// SIMATIC STEP 7 (V5.x) project PlcTornioFisher
// CPU: PLC317-2DP
// station: Hardware
// station: SINUMERIK
// station: P_ADR_BUS
// program: Programma S7(1)
// program: gp8x0d - PLC-Basicprogram-800Dsl 02.07.06 11/08/15
// program: SINAMICS_In_NCU_720
// program: SINAMICS_NX15_SINUMERIK

SYMBOL_TABLE
"ALMSG_DB"	DB 2	UDT 2	// Interface for Alarms & Messages
"gp_par"	DB 7	FB 1	// Parameters for Baseprogram
"NC"	DB 10	UDT 10	// Interface NC
"BAG"	DB 11	UDT 11	// Interface for BAG
"PI"	DB 16	DB 16	// Datainterface PI-Services
"SPL"	DB 18	DB 18	// SPL dataarea
"MMC"	DB 19	UDT 19	// Interface MMC-Signals
"Opzioni"	DB 20	UDT 20	// Opzioni macchina
"Canale1"	DB 21	UDT 21	// Interfaccia per Canale 1
"Canale2"	DB 22	UDT 21	// Interfaccia per Canale 2
"Canale3"	DB 23	UDT 21	// Interfaccia per Canale 3
"Canale4"	DB 24	UDT 21	// Interfaccia per Canale 4
"Asse_X1"	DB 31	UDT 31	// Interfaccia per Asse X1
"Asse_Z1"	DB 32	UDT 31	// Interfaccia per Asse Z1
"Asse_A"	DB 33	UDT 31	// Interfaccia per Asse A
"Asse_X2"	DB 34	UDT 31	// Interfaccia per Asse X2
"Asse_Z2"	DB 35	UDT 31	// Interfaccia per Asse Z2
"Asse_B"	DB 36	UDT 31	// Interfaccia per Asse B
"Asse_W"	DB 37	UDT 31	// Interfaccia per Asse W
"Asse_SP"	DB 38	UDT 31	// Interfaccia per Mandrino
"TMLoadIF"	DB 71	UDT 71	// Interface for Loading Station (Toolmanag.)
"TMSpindleIF"	DB 72	UDT 72	// Interface Spindle for Toolmanagment
"TMRevIF"	DB 73	UDT 73	// Interface Revolver (Toolmanagment)
"DB77"	DB 77	UDT 77	// SIEMENS
"CtrlE"	DB 1000	DB 1000	// Interface Ctrl-Energy
"SentronPac"	DB 1001	DB 1001	// Interface SentronPac
"RUN_UP"	FB 1	FB 1	// Startup Baseprogram
"GET"	FB 2	FB 2	// read NC Variable
"PUT"	FB 3	FB 3	// write NC Variable
"PI_SERV"	FB 4	FB 4	// PI-Services 1
"GETGUD"	FB 5	FB 5	// read GUD-Variable
"PI_SERV2"	FB 7	FB 7	// PI-Services 2
"M2N"	FB 9	FB 9	// Several OPs/NCUs
"SI_Relais"	FB 10	FB 10	// Safety Integrated: Relais
"SI_BrakeTest"	FB 11	FB 11	// Safety Integrated: Brake Test
"Diagnose"	FB 29	FB 29	// Signal recorder and data trigger diagnostics
"GP_HP"	FC 2	FC 2	// cyclic Baseprogram
"GP_PRAL"	FC 3	FC 3	// alarmtriggered Baseprogram
"GP_DIAG"	FC 5	FC 5	// Diagnosis alarm and Modul failure
"TM_TRANS2"	FC 6	FC 6	// Transfer for Toolmanagment (Multitool)
"TM_REV"	FC 7	FC 7	// Transfer for Revolverchange
"TM_TRANS"	FC 8	FC 8	// Transfer for Toolmanagment
"ASUP"	FC 9	FC 9	// asynchronous Subprograms
"AL_MSG"	FC 10	FC 10	// Alarms & Messages
"BHGDisp"	FC 13	FC 13	// Displaycontrol for Handheld Unit
"YDelta"	FC 17	FC 17	// Y / Delta Control
"SpinCtrl"	FC 18	FC 18	// Spindlecontrol / Part-, Positioning-axis
"MCP_IFM"	FC 19	FC 19	// MCP-Signals to Interface, Variant M
"Transfer"	FC 21	FC 21	// Quick Datachannel
"TM_DIR"	FC 22	FC 22	// Directioncontrol for Toolmanagment Mag.
"MCP_IFM2"	FC 24	FC 24	// MCP-Signals to Interface, Variant small
"MCP_IFT"	FC 25	FC 25	// MCP-Signals to Interface, Variant T
"HPU_MCP"	FC 26	FC 26	// MCP-Signals of PHG to Interface
"iNO_Emergenza_C1"	I 32.0	BOOL	// Emergenza ripristinata (Canale 1)
"iAux_ON(NC)"	I 32.1	BOOL	// Ausiliari inseriti (NC)
"iMax_Temp_AR"	I 32.2	BOOL	// Max temperatura alimentatore assi e mandrino
"iAR_Pronto"	I 32.3	BOOL	// Alimentatore assi e mandrino pronto
"iMax_Temp_Sorvegl"	I 32.4	BOOL	// Max temperatura modulo di sorveglianza
"iSorvegl_Pronto"	I 32.5	BOOL	// Modulo di sorveglianza pronto
"iPuls_Consenso"	I 32.6	BOOL	// 20SB1 - 20KA1 - Pulsante di consenso
"iAux_ON(NA)"	I 32.7	BOOL	// 18KA1 - Ausiliari inseriti (NA)
"iQM_Pompa_Idraul"	I 33.0	BOOL	// 3QM1 - Magnetotermico Pompa idraulica
"iQM_Sist_Serraggio"	I 33.1	BOOL	// 3QM2 - Magnetotermico Sistema di serraggio
"iQM_Controllo_Utensili"	I 33.2	BOOL	// 3QM3 - Magnetotermico Dispositivo Controllo Utensili
"iQM_Ventilat_Mandrino"	I 33.3	BOOL	// 3QM4 - MagnetotermicoVentilatore Mandrino
"iQF_Trasformatore"	I 33.4	BOOL	// 4QF1 - Magnetotermico Protezione trasformatore
"iQF_Utenze_110Vac"	I 33.5	BOOL	// 4QF2 - Magnetotermico Protezione Utenze a 110 Vac
"iQF_Prese_Illuminaz_QE"	I 33.6	BOOL	// 4QF3+4QF4 - Magnetot. Protez. Presa Pulpito e Q.E. +Illuminaz. Quadro
"iQF_Montronix"	I 33.7	BOOL	// 4QF5 - Magnetotermico Protezione Alimentazione Montronix
"iQF_Alim_24V_Uscite"	I 34.0	BOOL	// 5QF1 - Magnetotermico Protezione Sitop 24V Uscite
"iQF_Illuminaz_Macch"	I 34.1	BOOL	// 5QF2 - Magnetotermico Protezione Illuminaz. Macchina
"iQF_24V_UsciteSempreAlim"	I 34.2	BOOL	// 5QF3 - Magnetotermico Protezione Uscite PLC sempre alimentate
"iQF_24V_Uscite_Sezionate"	I 34.3	BOOL	// 5QF4 - Magnetotermico Protezione Uscite PLC sezionate
"iQF_Marposs"	I 34.4	BOOL	// 5QF6 - Magnetotermico Protezione Marposs
"iQF_Elettronica_CN"	I 34.5	BOOL	// 5QF7 - Magnetotermico Protezione Elettronica CN
"iQF_Condizionatori"	I 34.6	BOOL	// 6QF1+6QF2 Magnetot. Protez. condizionatori e trasformatore condizionatori
"iQF_Freno_Mandrino"	I 34.7	BOOL	// 12QF1 - Magnetotermico Protezione Freno Mandrino
"iQF_Uscite_Caricatore"	I 35.0	BOOL	// 5QF8 - Magnetotermico Protezione Uscite Caricatore
"iQF_Ingressi_PLC"	I 35.1	BOOL	// 5QF5 - Magnetotermico Protezione Alimentazione Ingressi PLC
"iBP35.2"	I 35.2	BOOL	// BP35.2 - Pressostato Blocco utensili sistema B serrato
"iBP35.3"	I 35.3	BOOL	// BP35.3 - Pressostato Blocco utensili sistema B disserrato
"iBP35.4"	I 35.4	BOOL	// BP35.4 - Pressostato Blocco utensili sistema A serrato
"iBP35.5"	I 35.5	BOOL	// BP35.5 - Pressostato Blocco utensili sistema A disserrato
"iBQ_Rip_Renishaw_Chiuso"	I 35.6	BOOL	// BP35.6 - Proximity Riparo controllo utensili chiuso
"iBQ_Rip_Renishaw_Aperto"	I 35.7	BOOL	// BP35.7 - Proximity Riparo controllo utensili aperto
"iNO_Emergenza_C2"	I 36.0	BOOL	// Emergenza ripristinata (Canale 2)
"iSA_AUTO"	I 36.1	BOOL	// SA36.1 - Selettore Funzionamento automatico
"iBQ36.3"	I 36.3	BOOL	// BQ36.3 - Proximity Braccio di misura in posiz. di misura
"iBQ36.4"	I 36.4	BOOL	// BQ36.4 - Proximity Braccio di misura a riposo
"iBP36.5"	I 36.5	BOOL	// BQ36.5 - Pressostato Filtro serraggio OK
"iKM_Pompa_Oleod_Inserita"	I 36.6	BOOL	// 51KM1 - Pompa oleodinamica inserita
"E36.7"	I 36.7	BOOL	// Disponibile
"iSQ_Oltrecorsa_X1+"	I 37.0	BOOL	// SQ37.0 - Finecorsa Oltrecorsa asse X1+
"iSQ_Oltrecorsa_X1-"	I 37.1	BOOL	// SQ37.1 - Finecorsa Oltrecorsa asse X1-
"iSQ_Ref_X1"	I 37.2	BOOL	// SQ37.2 - Finecorsa Punto di riferimento asse X1
"iSQ_Oltrecorsa_Z1+"	I 37.3	BOOL	// SQ37.3 - Finecorsa Oltrecorsa asse Z1+
"iSQ_Oltrecorsa_Z1-"	I 37.4	BOOL	// SQ37.4 - Finecorsa Oltrecorsa asse Z1-
"iSQ_Ref_Z1"	I 37.5	BOOL	// SQ37.5 - Finecorsa Punto di riferimento asse Z1
"iSQ_Oltrecorsa_X2+"	I 37.6	BOOL	// SQ37.6 - Finecorsa Oltrecorsa asse X2+
"iSQ_Oltrecorsa_X2-"	I 37.7	BOOL	// SQ37.7 - Finecorsa Oltrecorsa asse X2-
"iSQ_Ref_X2"	I 38.0	BOOL	// SQ38.0 - Finecorsa Punto di riferimento asse X2
"iSQ_Oltrecorsa_Z2+"	I 38.1	BOOL	// SQ38.1 - Finecorsa Oltrecorsa asse Z2+
"iSQ_Oltrecorsa_Z2-"	I 38.2	BOOL	// SQ38.2 - Finecorsa Oltrecorsa  asse Z2-
"iSQ_Ref_Z2_A"	I 38.3	BOOL	// SQ38.3 - Finecorsa Punto di riferimento A asse Z2
"iSQ_Ref_Z2_B"	I 38.4	BOOL	// SQ38.4 - Finecorsa Punto di riferimento B asse Z2
"iSQ_Cann_Avanz"	I 38.5	BOOL	// SQ38.5 - Finecorsa Posizione Cannotto Avanzato
"iSQ_Cann_Richiam"	I 38.6	BOOL	// SQ38.6 - Finecorsa Posizione Cannotto Richiamato
"iSQ_Oltrecorsa_W+"	I 38.7	BOOL	// SQ38.7 - Finecorsa Oltrecorsa+ Contropunta
"iSQ_Oltrecorsa_W-"	I 39.0	BOOL	// SQ39.0 - Finecorsa Oltrecorsa- Contropunta
"iSQ_Ref_W"	I 39.1	BOOL	// SQ39.1 - Finecorsa Punto di riferimento Contropunta
"iSQ_Oltrecorsa_W_Addiz"	I 39.2	BOOL	// SQ39.2 - Finecorsa Oltrecorsa addizionale Contropunta
"iSQ_Rapido_W"	I 39.3	BOOL	// SQ39.3 - Finecorsa Rapido contropunta
"iBP39.4"	I 39.4	BOOL	// BP39.4 - Pressostato Pompa prevalenza alta pressione OK
"i19SQ1"	I 39.5	BOOL	// 19SQ1 - Porta paraspruzzi chiave inserita
"iBP39.6"	I 39.6	BOOL	// BP39.6 - Pressostato Pompa idraulica filtra olio OK
"i19KA2_Porta_Bloccata"	I 39.7	BOOL	// 19KA2 - Finecorsa di sicurezza Porta paraspruzzi chiusa
"iBL40.0"	I 40.0	BOOL	// BL40.0 - Livellostato Lubrificazione ad impulsi
"iBP40.1"	I 40.1	BOOL	// BP40.1 - Pressostato Lubrificazione ad impulsi
"iBQ40.2"	I 40.2	BOOL	// BQ40.2 - Proximity  Riparo scorrevole chiuso
"iBQ40.3"	I 40.3	BOOL	// BQ40.3 - Proximity  Riparo scorrevole aperto
"iBL40.4"	I 40.4	BOOL	// BL40.4 - Livellostato Livello olio sistema serraggio
"iBT40.5"	I 40.5	BOOL	// BT40.5 - Termostato Quadro elettrico
"iBP40.6"	I 40.6	BOOL	// BP40.6 - Pressostato Cilindro di serraggio tirante 1 avanzato
"iBP40.7"	I 40.7	BOOL	// BP40.7 - Pressostato Cilindro di serraggio tirante 1 richiamato
"iBQ41.0"	I 41.0	BOOL	// BQ41.0 - Proximity Cilindro di serraggio tirante 1 in zona di serraggio
"iBQ41.1"	I 41.1	BOOL	// BQ41.1 - Proximity Cilindro di serraggio tirante 1 in zona finale
"iBP41.2"	I 41.2	BOOL	// BP41.2 - Pressostato Cannotto Avanti in pressione
"iSQ_Cannotto_Avanti"	I 41.3	BOOL	// SQ41.3 - Finecorsa Cannotto Avanzato
"iSQ_Cannotto_Indietro"	I 41.4	BOOL	// SQ41.4 - Finecorsa Cannotto Richiamata
"iBP_Controtesta_Serrata"	I 41.5	BOOL	// BP41.5 - Pressostato Controtesta serrata
"iBP_Controtesta_Lubr_OK"	I 41.6	BOOL	// BP41.6 - Pressostato Controtesta pressione lubrificazione OK
"i51KM5"	I 41.7	BOOL	// 51KM5 - Ventilatore mandrino in marcia
"E42.0"	I 42.0	BOOL	// Disponibile
"E42.1"	I 42.1	BOOL	// Disponibile
"E42.2"	I 42.2	BOOL	// Disponibile
"E42.3"	I 42.3	BOOL	// Disponibile
"E42.4"	I 42.4	BOOL	// Disponibile
"E42.5"	I 42.5	BOOL	// Disponibile
"iBQ_TorrA_Bloccata"	I 42.6	BOOL	// BQ42.6 - Proximity Torretta A bloccata
"iBQ_TorrA_Sbloccata"	I 42.7	BOOL	// BQ42.7 - Proximity Torretta A sbloccata
"E43.0"	I 43.0	BOOL	// Disponibile
"E43.1"	I 43.1	BOOL	// Disponibile
"E43.2"	I 43.2	BOOL	// Disponibile
"E43.3"	I 43.3	BOOL	// Disponibile
"E43.4"	I 43.4	BOOL	// Disponibile
"E43.5"	I 43.5	BOOL	// Disponibile
"iBQ_TorrB_Bloccata"	I 43.6	BOOL	// BQ43.6 - Proximity Torretta B bloccata
"iBQ_TorrB_Sbloccata"	I 43.7	BOOL	// BQ43.7 - Proximity Torretta B sbloccata
"E44.0"	I 44.0	BOOL	// Disponibile
"E44.1"	I 44.1	BOOL	// Disponibile
"E44.2"	I 44.2	BOOL	// Disponibile
"E44.3"	I 44.3	BOOL	// Disponibile
"E44.4"	I 44.4	BOOL	// Disponibile
"E44.5"	I 44.5	BOOL	// Disponibile
"E44.6"	I 44.6	BOOL	// Disponibile
"E44.7"	I 44.7	BOOL	// Disponibile
"iPL_Sist_Aux_Inser"	I 45.0	BOOL	// Caricatore - Sistema Aux Inserito
"iPL_Ciclo_Auto"	I 45.1	BOOL	// Caricatore - Ciclo Automatico in corso
"iPL_Portale_Inserito"	I 45.2	BOOL	// Caricatore - Almeno un portale inserito
"iPL_Prelievo_OK"	I 45.3	BOOL	// Caricatore - Prelievo avvenuto
"iPL_Cons_Sblocc_Pz"	I 45.4	BOOL	// Caricatore - Consenso sbloccaggio pezzo
"iPL_Deposito_OK"	I 45.5	BOOL	// Caricatore - Deposito avvenuto
"iPL_Cons_Bloc_Pz"	I 45.6	BOOL	// Caricatore - Consenso bloccaggio pezzo
"iPL_Fuori_Ingombro"	I 45.7	BOOL	// Caricatore - Fuori ingombro
"iPL_Cambio_Tipo"	I 46.0	BOOL	// Caricatore - Cambo Tipo
"iPL_Gest_Auto_Isola"	I 46.1	BOOL	// Caricatore - Gestione automatica isola
"iPL_Cod_Tipo_Strobe"	I 46.2	BOOL	// Caricatore - Codifica Tipo strobe
"iPL_Cod_Tipo_Bit1"	I 46.3	BOOL	// Caricatore - Codifica Tipo bit 1
"iPL_Cod_Tipo_Bit2"	I 46.4	BOOL	// Caricatore - Codifica Tipo bit 2
"iPL_Cod_Tipo_Bit3"	I 46.5	BOOL	// Caricatore - Codifica Tipo bit 3
"iPL_Cod_Tipo_Bit4"	I 46.6	BOOL	// Caricatore - Codifica Tipo bit 4
"iPL_Cod_Tipo_Parità"	I 46.7	BOOL	// Caricatore - Codifica Tipo parità pari
"iPL_Cons_Prebloc_Pz"	I 47.0	BOOL	// Caricatore - Consenso prebloccaggio pezzo
"iPL_Cons_Prel_Grezzo"	I 47.1	BOOL	// Caricatore - Richiestra prelievo grezzo
"iPL_Disp1"	I 47.2	BOOL	// Caricatore - Disponibile
"iPL_Disp2"	I 47.3	BOOL	// Caricatore - Disponibile
"iMarposs_Dati_Validi"	I 47.4	BOOL	// Marposs - Dati Validi (come da schema elettrico)
"E47.5"	I 47.5	BOOL	// Disponibile
"E47.6"	I 47.6	BOOL	// Disponibile
"E47.7"	I 47.7	BOOL	// Disponibile
"iMarposs_Misura_1"	I 48.0	BOOL	// Marposs -N° misura 1
"iMarposs_Misura_2"	I 48.1	BOOL	// Marposs -N° misura 2
"iMarposs_Misura_4"	I 48.2	BOOL	// Marposs -N° misura 4
"iMarposs_Misura_8"	I 48.3	BOOL	// Marposs -N° misura 8
"iMarposs_Misura_10"	I 48.4	BOOL	// Marposs -N° misura 10
"iMarposs_Misura_20"	I 48.5	BOOL	// Marposs -N° misura 20
"iMarposs_Misura_40"	I 48.6	BOOL	// Marposs -N° misura 40
"iMarposs_Misura_80"	I 48.7	BOOL	// Marposs -N° misura 80
"iMarposs_Valore_1"	I 49.0	BOOL	// Marposs -Valore 1
"iMarposs_Valore_2"	I 49.1	BOOL	// Marposs -Valore 2
"iMarposs_Valore_4"	I 49.2	BOOL	// Marposs -Valore 4
"iMarposs_Valore_8"	I 49.3	BOOL	// Marposs -Valore 8
"iMarposs_Valore_10"	I 49.4	BOOL	// Marposs -Valore 10
"iMarposs_Valore_20"	I 49.5	BOOL	// Marposs -Valore 20
"iMarposs_Valore_40"	I 49.6	BOOL	// Marposs -Valore 40
"iMarposs_Valore_80"	I 49.7	BOOL	// Marposs -Valore 80
"iMarposs_Valore_100"	I 50.0	BOOL	// Marposs -Valore 100
"iMarposs_Valore_200"	I 50.1	BOOL	// Marposs -Valore 200
"iMarposs_Valore_400"	I 50.2	BOOL	// Marposs -Valore 400
"iMarposs_Valore_800"	I 50.3	BOOL	// Marposs -Valore 800
"iMarposs_Valore_1000"	I 50.4	BOOL	// Marposs -Valore 1000
"iMarposs_Segno 1=-"	I 50.5	BOOL	// Marposs - Segno 1=""-""
"iMarposs_Parità"	I 50.6	BOOL	// Marposs - Parità
"iMarposs_Dati_Pronti"	I 50.7	BOOL	// Marposs - Dati pronti
"iMarposs_Scarto_Irrecup"	I 51.0	BOOL	// Marposs - Scarto irrecuperabile
"iMarposs_Correzione"	I 51.1	BOOL	// Marposs - Correzione
"iMarposs_Correz_Indietro"	I 51.2	BOOL	// Marposs - Correzione indietro
"iMarposs_Misura_OK"	I 51.3	BOOL	// Marposs - Misura buona
"iMarposs_Correz_Avanti"	I 51.4	BOOL	// Marposs - Correzione avanti
"iMarposs_Dati_Validi_New"	I 51.5	BOOL	// Marposs - Dati Validi (come da sw PLC)
"iMarposs_Disp2"	I 51.6	BOOL	// Marposs - Disponibile
"iMarposs_Scarto_Recuper"	I 51.7	BOOL	// Marposs - Scarto recuperabile
"iBP_Lubrif_Z1_OK"	I 52.0	BOOL	// BP52.0 - Pressostato Sistema A asse Z OK
"iBP_Lubrif_X1_OK"	I 52.1	BOOL	// BP52.1 - Pressostato Sistema A asse X OK
"iBP_Lubrif_Z2_OK"	I 52.2	BOOL	// BP52.2 - Pressostato Sistema B asse X OK
"iBP_Lubrif_X2_OK"	I 52.3	BOOL	// BP52.3 - Pressostato Sistema B asse Z OK
"iBP_Lubrif_Serrag_OK"	I 52.4	BOOL	// BP52.4 - Pressostato Mandrino di serraggio OK
"iBT_Sist_Serraggio_OK"	I 52.5	BOOL	// BT52.5 - Temperatura sistema di serraggio OK
"E52.6"	I 52.6	BOOL	// Disponibile
"E52.7"	I 52.7	BOOL	// Disponibile
"iLiv_Olio_Sblocco_Ciclo"	I 53.0	BOOL	// Livello olio - Sblocco ciclo
"iLiv_Olio_Prelim_Liv_Min"	I 53.1	BOOL	// Livello olio - Allarme preliminare di livello minimo
"iLiv_Olio_All_Colaggio"	I 53.2	BOOL	// Livello olio - Allarme di colaggio
"iSblocco_Pompa_Oleod_Ins"	I 53.3	BOOL	// 60KA1 - Controllo livello olio sblocco pompa oleodinamica inserito
"iMonit_Manut_Sist_Ins"	I 53.4	BOOL	// Monitor Manutenzione - Sistema inserito
"iMonit_Manut_Attesa"	I 53.5	BOOL	// Monitor Manutenzione - Attesa di manutenzione
"iMonit_Manut_Non_Eseguit"	I 53.6	BOOL	// Monitor Manutenzione - Manutenzione non eseguita
"iMonit_Manut_Fermata"	I 53.7	BOOL	// Monitor Manutenzione - Fermata macchina
"iBP_Aria_OK"	I 54.0	BOOL	// BP54.0 - Pressione aria compressa OK
"iBP_Refriger_OK"	I 54.1	BOOL	// BP54.1 - Pressione refrigerante OK
"iMontrA_Disp"	I 54.2	BOOL	// Montronix A - Disponibile
"iMontrA_Rottura_Utensile"	I 54.3	BOOL	// Montronix A - Rottura Utensile
"iMontrA_Usura_Utensile"	I 54.4	BOOL	// Montronix A - Usura Utensile
"iMontrA_In_Funzione"	I 54.5	BOOL	// Montronix A - In funzione
"iMontrA_Mancanza_Utens"	I 54.6	BOOL	// Montronix A - Mancanza Utensile
"iMontrA_Collisione"	I 54.7	BOOL	// Montronix A - Sistema A collisione
"iMontrB_Disp"	I 55.0	BOOL	// Montronix B - Disponibile
"iMontrB_Rottura_Utensile"	I 55.1	BOOL	// Montronix B - Rottura Utensile
"iMontrB_Usura_Utensile"	I 55.2	BOOL	// Montronix B - Usura Utensile
"iMontrB_In_Funzione"	I 55.3	BOOL	// Montronix B - In funzione
"iMontrB_Mancanza_Utens"	I 55.4	BOOL	// Montronix B - Mancanza Utensile
"iMontrB_Collisione"	I 55.5	BOOL	// Montronix B - Sistema A collisione
"E55.6"	I 55.6	BOOL	// Disponibile
"E55.7"	I 55.7	BOOL	// Disponibile
"mAll_700000"	I 72.0	BOOL	// Vita Utensile Esaurita
"mAll_700001"	I 72.1	BOOL	// ERR 7001 TENSIONE DI COM. NON INSERITA
"mAll_700002"	I 72.2	BOOL	// ERR 7002 POMPA IDRAUL. NON FUNZIONA
"mAll_700003"	I 72.3	BOOL	// ERR 7003 INTERR. A CHIAVE  MODO AUTOM.
"mAll_700007"	I 72.7	BOOL	// ERR 7007 MOVIMENTO ATT. A PORTA APERTA
"mAll_700016"	I 74.0	BOOL	// ERR 7016 MANDR.1 MOTORE,REGOLATORE CALDO
"mAll_700017"	I 74.1	BOOL	// ERR 7017 MANDR.1 COPPA MOTRICE > 90%
"mAll_700018"	I 74.2	BOOL	// ERR 7018 MANDR.1 NON PRONTO
"mAll_700019"	I 74.3	BOOL	// ERR 7019 MANDR.1 GUASTO VENTILATORE
"mAll_700020"	I 74.4	BOOL	// ERR 7020 MANDR.1 MONITORE N EFF<N MIN
"mAll_700021"	I 74.5	BOOL	// ERR 7021 MANDR.1 MONITORE N EFF=N NOM
"mAll_700022"	I 74.6	BOOL	// ERR 7022 MANDR.1 MONITORE DURATA INSERZ.
"mAll_700023"	I 74.7	BOOL	// ERR 7023 MANDR.1 CONFUSIONE DI VELOCITA
"mAll_700024"	I 75.0	BOOL	// ERR 7024 COM.AVANZ.MC MOTORE NON PRONTO
"mAll_700025"	I 75.1	BOOL	// ERR 7025 COM.AVANZ.MC ASSI NON PRONTI
"mAll_700027"	I 75.3	BOOL	// ERR 7027 COM.AVANZ.MC FINE CORSA ASSE X1
"mAll_700028"	I 75.4	BOOL	// ERR 7028 MC MOTORE ASSE X1 ECC.DI TEMP.
"mAll_700030"	I 75.6	BOOL	// ERR 7030 COM.AVANZ.MC FINE CORSA ASSE Z1
"mAll_700031"	I 75.7	BOOL	// ERR 7031 MC MOTORE ASSE Z1 ECC.DI TEMP.
"mAll_700100"	I 76.0	BOOL	// ERR 7032 MC MOTORE X1 NON SULL'ORIGINE
"mAll_700101"	I 76.1	BOOL	// ERR 7033 COM.AVANZ.MC FINE CORSA ASSE X2
"mAll_700102"	I 76.2	BOOL	// ERR 7034 MC MOTORE ASSE X2 ECC.DI TEMP.
"mAll_700104"	I 76.4	BOOL	// ERR 7036 COM.AVANZ.MC FINE CORSA ASSE Z2
"mAll_700105"	I 76.5	BOOL	// ERR 7037 MC MOTORE ASSE Z2 ECC.DI TEMP.
"mAll_700106"	I 76.6	BOOL	// ERR 7038 MC MOTORE X2 NON SULL'ORIGINE
"mAll_700107"	I 76.7	BOOL	// ERR 7039 COM.AVANZ.MC FINE CORSA ASSE W
"mAll_700108"	I 77.0	BOOL	// ERR 7040 MC MOTORE ASSE W ECC.DI TEMP.
"mAll_700110"	I 77.2	BOOL	// ERR 7042 COM.AVANZ.MC FINE CORSA ASSE Q
"mAll_700111"	I 77.3	BOOL	// ERR 7043 MC MOTORE ASSE Q ECC.DI TEMP.
"mAll_700114"	I 77.6	BOOL	// ERR 7046 MC MOTORE ASSE C ECC.DI TEMP.
"mAll_700116"	I 78.0	BOOL	// ERR 7048 ANOMALIA DI LUBRIFICAZIONE
"mAll_700117"	I 78.1	BOOL	// ERR 7049 LUBRIFIC.  LIVELLO OLIO BASSO
"mAll_700118"	I 78.2	BOOL	// ERR 7050 ALTA PRESSIONE NON IN ORDINE
"mAll_700119"	I 78.3	BOOL	// ERR 7051 SEQ CONTROTESTA NON SBLOCCATA
"mAll_700120"	I 78.4	BOOL	// ERR 7052 SEQ CONTROTESTA NON BLOCCATA
"mAll_700121"	I 78.5	BOOL	// ERR 7053 CONTROTESTA NON BLOCC./SBLOCC.
"mAll_700122"	I 78.6	BOOL	// ERR 7054 TASTO DI RESET AZION. (C.TESTA)
"mAll_700123"	I 78.7	BOOL	// ERR 7055 CANNOT. DAVANTI A C.TESTA SBLOC
"mAll_700127"	I 79.3	BOOL	// ERR 7059 MC MOTORE Q  CONF. ORIGINE SCOR
"mAll_700128"	I 79.4	BOOL	// ERR 7060 MC MOTORE Z2 CONF. ORIGINE SCOR
"mAll_700129"	I 79.5	BOOL	// ERR 7061 MC MOTORE X1 CONF. ORIGINE SCOR
"mAll_700130"	I 79.6	BOOL	// ERR 7062 MC MOTORE Z1 ORIGINE N.ABBORDAT
"mAll_700131"	I 79.7	BOOL	// ERR 7063 MC MOTORE X2 ORIGINE N.ABBORDAT
"mAll_700200"	I 80.0	BOOL	// ERR 7064 MC MOTORE Z2 ORIGINE N.ABBORDAT
"mAll_700201"	I 80.1	BOOL	// ERR 7065 MC MOTORE W  ORIGINE N.ABBORDAT
"mAll_700202"	I 80.2	BOOL	// ERR 7066 MC MOTORE Q  ORIGINE N.ABBORDAT
"mAll_700204"	I 80.4	BOOL	// ERR 7068 MC MOTORE Y1 ORIGINE N.ABBORDAT
"mAll_700206"	I 80.6	BOOL	// ERR 7070 ARRESTO MANDRINO+AVANZAMENTO
"mAll_700207"	I 80.7	BOOL	// ERR 7071 ARRESTO AVANZAMENTO
"mAll_700208"	I 81.0	BOOL	// ERR 7072 MANDR.1 ASSE C NON ACCOPPIATO
"mAll_700209"	I 81.1	BOOL	// ERR 7073 MANDR.1 ASSE C NON STACCATO
"mAll_700210"	I 81.2	BOOL	// ERR 7074 CONTR. LIVELLO OLIO  N.SBLOCC.
"mAll_700211"	I 81.3	BOOL	// ERR 7075 CONTR. LIV.OLIO IDR. N.SBLOCC.
"mAll_700212"	I 81.4	BOOL	// ERR 7076 MANDR.1 ASSE C NON STACCATO
"mAll_700213"	I 81.5	BOOL	// ERR 7077 MIS.UT. SEQ  APRIRE RIPARO
"mAll_700214"	I 81.6	BOOL	// ERR 7078 MIS.UT. SEQ  CHIUDERE RIPARO
"mAll_700215"	I 81.7	BOOL	// ERR 7079 MIS.UT. SEQ  RICHIAMO BRACCIO
"mAll_700216"	I 82.0	BOOL	// ERR 7080 MIS.UT. SEQ  ABBORDAM. BRACCIO
"mAll_700217"	I 82.1	BOOL
"mAll_700218"	I 82.2	BOOL	// ERR 7082 MIS.UT. BRACCIO IN POS.INDEF.
"mAll_700219"	I 82.3	BOOL	// ERR 7083 MIS.UT. PEZZO NON DISSERRATO
"mAll_700220"	I 82.4	BOOL	// ERR 7084 TRASP.TRUCIOLI SOVRACCAR.ELETTR
"mAll_700221"	I 82.5	BOOL	// ERR 7085 TRASP.TRUCIOLI SOVRACCAR.MECCAN
"mAll_700222"	I 82.6	BOOL	// ERR 7086 ARMADIO ELETTR.  ECC.DI TEMPER.
"mAll_700223"	I 82.7	BOOL	// ERR 7087 FILTRAOLIO INTASATO
"mAll_700224"	I 83.0	BOOL	// ERR 7088 LIV.OLIO  ALLARME DI PERDITA
"mAll_700225"	I 83.1	BOOL	// ERR 7089 LIV.OLIO  PREALLARME DI MIN.
"mAll_700226"	I 83.2	BOOL	// ERR 7090 MANDR.1 BLOCCATO
"mAll_700228"	I 83.4	BOOL	// ERR 7092 MANDRINO COMMUTAZIONE BLOCCATA
"mAll_700229"	I 83.5	BOOL	// ERR 7093 MANDRINO TIME OUT COMMUTAZIONE
"mAll_700230"	I 83.6	BOOL	// ERR 7094 MANDR.1  USURA SPAZZOLE
"mAll_700300"	I 84.0	BOOL	// ERR 7100 CIL.1  SERRAGGIO CONTR.SEQU.
"mAll_700301"	I 84.1	BOOL	// ERR 7101 CIL.1  DISSERR. CONTR.SEQU.
"mAll_700302"	I 84.2	BOOL	// ERR 7102 CIL.1  MANOCONTATTO SEGN.INDEF.
"mAll_700303"	I 84.3	BOOL	// ERR 7103 CIL.1  FINE CORSA SEGN.INDEF.
"mAll_700305"	I 84.5	BOOL	// ERR 7105 CIL.2  SERRAGGIO CONTR.SEQU.
"mAll_700306"	I 84.6	BOOL	// ERR 7106 CIL.2  DISSERR. CONTR.SEQU.
"mAll_700307"	I 84.7	BOOL	// ERR 7107 CIL.2  MANOCONTATTO SEGN.INDEF.
"mAll_700308"	I 85.0	BOOL	// ERR 7108 COL.2  FINE CORSA SEGN.INDEF.
"mAll_700310"	I 85.2	BOOL	// ERR 7110 CANNOTTO AVANTI  CONTR.DI SEQU.
"mAll_700311"	I 85.3	BOOL	// ERR 7111 CANNOTTO INDIETRO CONTR. SEQU.
"mAll_700312"	I 85.4	BOOL	// ERR 7112 CANNOT. AVANTI A META CONTR.SEQ
"mAll_700313"	I 85.5	BOOL	// ERR 7113 CANNOT. INDIETRO A META  C.SEQU
"mAll_700314"	I 85.6	BOOL	// ERR 7114 CANNOTTO C.TESTA POS. INDEF.
"mAll_700315"	I 85.7	BOOL	// ERR 7115 START CN EFF. SOLO PER CANALE 1
"mAll_700316"	I 86.0	BOOL	// ERR 7116 START CN EFF. SOLO PER CANALE 2
"mAll_700317"	I 86.1	BOOL	// ERR 7117 START CN EFF. SOLO PER CANALE 3
"mAll_700318"	I 86.2	BOOL	// ERR 7118 START CN EFF. SOLO PER CANALE 4
"mAll_700320"	I 86.4	BOOL	// ERR 7120 CIL.1 NON SERRATO
"mAll_700322"	I 86.6	BOOL	// ERR 7122 CIL.2 NON SERRATO
"mAll_700324"	I 87.0	BOOL	// ERR 7124 CANNOT. C.TESTA NON SERRATO
"mAll_700326"	I 87.2	BOOL	// ERR 7126 CONTROTESTA NON BLOCCATA
"mAll_700328"	I 87.4	BOOL	// ERR 7128 PEZZO NON FISSATO
"mAll_700330"	I 87.6	BOOL	// ERR 7130 TASTI MAN. DISP.DI SERR. BLOCC.
"mAll_700331"	I 87.7	BOOL	// ERR 7131 CAN.1 SERRAGGIO FUNZ.AUS. INACC
"mAll_700400"	I 88.0	BOOL	// ERR 7132 CAN.2 SERRAGGIO FUNZ.AUS. INACC
"mAll_700401"	I 88.1	BOOL	// ERR 7133 CAN.3 SERRAGGIO FUNY.AUS. INACC
"mAll_700402"	I 88.2	BOOL	// ERR 7134 PORTA PARASPRUZZI NON BLOCCATA
"mAll_700403"	I 88.3	BOOL	// ERR 7135 PORTA PARASPRUZZI NON SBLOCCATA
"mAll_700404"	I 88.4	BOOL	// ERR 7136 COM.AVANZ.MC FINE CORSA ASSE Y1
"mAll_700405"	I 88.5	BOOL	// ERR 7137 MC MOTORE ASSE Y1 ECC.DI TEMP.
"mAll_700406"	I 88.6	BOOL	// ERR 7138 COM.AVANZ.MC ASSE Y1 N.SBLOCC.
"mAll_700407"	I 88.7	BOOL	// ERR 7139 COM.AVANZ.MC ASSE Y1 N.BLOCC.
"mAll_700408"	I 89.0	BOOL	// ERR 7140 Torretta A NON BLOCCATA
"mAll_700411"	I 89.3	BOOL	// ERR 7143 Torretta A ROTAZIONE FERMATA
"mAll_700412"	I 89.4	BOOL	// ERR 7144 Torretta A MOVIMENTO FERMATO
"mAll_700413"	I 89.5	BOOL	// ERR 7145 Torretta A FERMATA
"mAll_700414"	I 89.6	BOOL	// ERR 7146 Torretta A ERRORE DI PARITA
"mAll_700415"	I 89.7	BOOL	// ERR 7147 Torretta A POSIZIONE SBAGLIATA
"mAll_700416"	I 90.0	BOOL	// ERR 7148 Torretta A ECCESSO DI TEMPERATURA
"mAll_700418"	I 90.2	BOOL	// ERR 7150 Torretta A SEQU. DI SBLOCCAGGIO
"mAll_700419"	I 90.3	BOOL	// ERR 7151 Torretta A SEQU. DI ROTAZIONE
"mAll_700420"	I 90.4	BOOL	// ERR 7152 Torretta A SEQU. DI POSIZIONAMENTO
"mAll_700421"	I 90.5	BOOL	// ERR 7153 Torretta A SEQU. DI BLOCCAGGIO
"mAll_700422"	I 90.6	BOOL	// ERR 7154 Torretta A NON BL0CCATA
"mAll_700423"	I 90.7	BOOL	// ERR 7155 Torretta A NON IN POSIZIONE
"mAll_700424"	I 91.0	BOOL	// ERR 7156 Torretta A CONTR. DEL SEGN. STROBE
"mAll_700426"	I 91.2	BOOL	// ERR 7158 Torretta A MANCA SENSO DI ROTAZ.
"mAll_700427"	I 91.3	BOOL	// ERR 7159 Torretta A T MANCA NELL'ATTREZ.MULT
"mAll_700428"	I 91.4	BOOL	// ERR 7160 Torretta B NON BLOCCATA
"mAll_700431"	I 91.7	BOOL	// ERR 7163 Torretta B ROTAZIONE FERMATA
"mAll_700500"	I 92.0	BOOL	// ERR 7164 Torretta B MOVIMENTO FERMATO
"mAll_700501"	I 92.1	BOOL	// ERR 7165 Torretta B FERMATA
"mAll_700502"	I 92.2	BOOL	// ERR 7166 Torretta B ERRORE DI PARITA
"mAll_700503"	I 92.3	BOOL	// ERR 7167 Torretta B POSIZIONE SBAGLATA
"mAll_700504"	I 92.4	BOOL	// ERR 7168 Torretta B ECCESSO DI TEMPERATURA
"mAll_700506"	I 92.6	BOOL	// ERR 7170 Torretta B SEQU. DI SBLOCCAGGIO
"mAll_700507"	I 92.7	BOOL	// ERR 7171 Torretta B SEQU. DI ROTAZONE
"mAll_700508"	I 93.0	BOOL	// ERR 7172 Torretta B SEQU. DI POSIZIONAMENTO
"mAll_700509"	I 93.1	BOOL	// ERR 7173 Torretta B SEQU. DI BLOCCAGGIO
"mAll_700510"	I 93.2	BOOL	// ERR 7174 Torretta B NON BLOCCATA
"mAll_700511"	I 93.3	BOOL	// ERR 7175 Torretta B NON IN POSIZIONE
"mAll_700512"	I 93.4	BOOL	// ERR 7176 Torretta B CONTR. DEL SEGN. STROBE
"mAll_700514"	I 93.6	BOOL	// ERR 7178 Torretta B MANCA SENSO DI ROTAZ.
"mAll_700515"	I 93.7	BOOL	// ERR 7179 Torretta B T MANCA NELL'ATTREZ.MULT
"mAll_700516"	I 94.0	BOOL	// ERR 7180 ROTTURA UTENSILE  SOVRACCARICO
"mAll_700517"	I 94.1	BOOL	// ERR 7181 ROTTURA UTENSILE  ROTTURA
"mAll_700518"	I 94.2	BOOL	// ERR 7182 ROTTURA UTENSILE  USURA
"mAll_700520"	I 94.4	BOOL	// ERR 7184 LUNETTA  SEQU. DI CHIUSURA
"mAll_700521"	I 94.5	BOOL	// ERR 7185 LUNETTA  SEQU. DI APERTURA
"mAll_700522"	I 94.6	BOOL	// ERR 7186 LUNETTA  SEQU. DI ACCOSTAMENTO
"mAll_700523"	I 94.7	BOOL	// ERR 7187 LUNETTA  SEQU. DI RICHIAMO
"mAll_700524"	I 95.0	BOOL	// ERR 7188 LUNETTA  LEVE IN POS. INDEF.
"mAll_700525"	I 95.1	BOOL	// ERR 7189 LUNETTA  SUPPORTO IN POS.INDEF.
"mAll_700526"	I 95.2	BOOL	// ERR 7190 LUNETTA  MANCA PRESSIONE
"mAll_700527"	I 95.3	BOOL	// ERR 7191 LUNETTA  COMANDO INACCETTABILE
"mAll_700528"	I 95.4	BOOL	// ERR 7192 MOTORE Q NELLA ZONA DI COLLIS.
"mAll_700600"	I 96.0	BOOL	// ERR 7200 MISURAZ. PEZZI: PEZZO SCARTO
"mAll_700601"	I 96.1	BOOL	// ERR 7201 CAN.1 CONTR. PROGR. N. IN ORD.
"mAll_700602"	I 96.2	BOOL	// ERR 7202 CAN.2 CONTR. PROGR. N. IN ORD.
"mAll_700603"	I 96.3	BOOL	// ERR 7203 CAN.3 CONTR. PROGR. N. IN ORD.
"mAll_700604"	I 96.4	BOOL	// ERR 7204 CAN.4 CONTR. ROGR. N. IN ORD.
"mAll_700605"	I 96.5	BOOL	// ERR 7205 PORTA PARASPR.  SEQU. DI CHIUS.
"mAll_700606"	I 96.6	BOOL	// ERR 7206 PORTA PARASPR.  SEQU. DI APERT.
"mAll_700607"	I 96.7	BOOL	// ERR 7207 PORTA PARASPR.  POS. INDEF
"mAll_700608"	I 97.0	BOOL	// ERR 7208 PORTA PARASPR.  PROTEZIONI
"mAll_700609"	I 97.1	BOOL	// ERR 7209 PORTA  ISTRUZ.IMPOSS. CAN.2
"mAll_700610"	I 97.2	BOOL	// ERR 7210 PORTA  ISTRUZ.IMPOSS. CAN.3
"mAll_700611"	I 97.3	BOOL	// ERR 7211 ERR.DI PROGRAM. SINCRON. CAN.1
"mAll_700612"	I 97.4	BOOL	// ERR 7212 ERR.DI PROGRAM. SINCRON. CAN.2
"mAll_700613"	I 97.5	BOOL	// ERR 7213 ERR DI PROGRAM. SINCRON. CAN.3
"mAll_700614"	I 97.6	BOOL	// ERR 7214 ERR.DI PROGRAM. SINCRON. CAN.4
"mAll_700615"	I 97.7	BOOL	// ERR 7215 PORTA PARASPR.  ISTRUZ.IMPOSS.
"mAll_700619"	I 98.3	BOOL	// ERR 7219 DURATA CICLO  DATI INACC. M868
"mAll_700620"	I 98.4	BOOL	// ERR 7220 MANUTENZ. MC NECESSARIA
"mAll_700621"	I 98.5	BOOL	// ERR 7221 MANUTENZ. PL NECESSARIA
"mAll_700622"	I 98.6	BOOL	// ERR 7222 ARRESTO CICLO DAL CONTAT.PEZZI
"mAll_700623"	I 98.7	BOOL	// ERR 7223 DURATA DEL CICLO SUPERATA
"mAll_700624"	I 99.0	BOOL	// ERR 7224 MANDR.1 BATTARELLA N.RICHIAMATA
"mAll_700625"	I 99.1	BOOL	// ERR 7225 MANDR.1 BATTARELLA NON ACCOSTAT
"mAll_700626"	I 99.2	BOOL	// ERR 7226 MANDR.1 BATTARELLA NON RICHIAM.
"mAll_700627"	I 99.3	BOOL	// ERR 7227 MANDR.1 ANOMALIA INGRANAGGIO
"mAll_700700"	I 100.0	BOOL	// ERR 7232 REFRIGER. POMPA NON INSERITA
"mAll_700701"	I 100.1	BOOL	// ERR 7233 REFRIGER. CONTROLLO LIVELLO
"mAll_700702"	I 100.2	BOOL	// ERR 7234 REFRIG. PREALL. DI LIV.MIN.
"mAll_700703"	I 100.3	BOOL	// ERR 7235 POMPA DI ALIM. NON INSERITA
"mAll_700704"	I 100.4	BOOL	// ERR 7236 REFRIGER. LIVELLO SERBATOIO
"mAll_700706"	I 100.6	BOOL	// ERR 7238 REFRIGER.  ALTA PRESSIONE
"mAll_700707"	I 100.7	BOOL	// ERR 7239 REFRIGER.  PASSAGGIO
"mAll_700708"	I 101.0	BOOL	// ERR 7240 UT.BLOC.A  NON FISSATO
"mAll_700709"	I 101.1	BOOL	// ERR 7241 UT.BLOC.A  SEQU.DI FISSAGGIO
"mAll_700710"	I 101.2	BOOL	// ERR 7242 UT.BLOC.A  SEQU.DI SBLOCC.
"mAll_700711"	I 101.3	BOOL	// ERR 7243 UT.BLOC.A  POS. INDEFINITA
"mAll_700712"	I 101.4	BOOL	// ERR 7244 UT.BLOC.A  COMANDO INACCETT.
"mAll_700713"	I 101.5	BOOL	// ERR 7245 UT.BLOC.B  NON FISSATO
"mAll_700714"	I 101.6	BOOL	// ERR 7246 UT.BLOC.B  SEQU.DI FISSAGGIO
"mAll_700715"	I 101.7	BOOL	// ERR 7247 UT.BLOC.B  SEQU.DI SBLOCC.
"mAll_700716"	I 102.0	BOOL	// ERR 7248 UT.BLOC.B  POS. INDEFINITA
"mAll_700717"	I 102.1	BOOL	// ERR 7249 UT.BLOC.B  COMANDO INACCETT.
"mAll_700718"	I 102.2	BOOL	// ERR 7250 MONITORE DI MAN.  SCARIC.PEZZO
"mAll_700719"	I 102.3	BOOL	// ERR 7251 MONIT.DI MAN. ESEG. MANUTENZ.
"mAll_700724"	I 103.0	BOOL	// ERR 7256 POMPA AD ALTA PRESS.  LIV.OLIO
"mAll_700725"	I 103.1	BOOL	// ERR 7257 POMPA A.PRESS.  ANOM.DI TEMPER.
"mAll_700726"	I 103.2	BOOL	// ERR 7258 POMPA A.PRESS.  ANOMALIA FILTRO
"mAll_700727"	I 103.3	BOOL	// ERR 7259 MANCA PRESS. DI ARIA COMPRESSA
"mAll_700728"	I 103.4	BOOL	// ERR 7260 MANCA PRESSIONE DI REFRIGERANTE
"mAll_700729"	I 103.5	BOOL	// ERR 7261 INTERR. AUTOM. NON IN ORDINE
"mAll_700730"	I 103.6	BOOL	// 6QF1+6QF2 Magnetot. Protez. condizionatori Intervenuto
"mAll_700731"	I 103.7	BOOL	// 12QF1 - Magnetotermico Protezione Freno Mandrino Intervenuto
"mAll_700800"	I 104.0	BOOL	// Magnetotermico Pompa idraulica Intervenuto - 3QM1
"mAll_700801"	I 104.1	BOOL	// 3QM2 - Magnetotermico Sistema di serraggio Intervenuto
"mAll_700802"	I 104.2	BOOL	// 3QM3 - Magnetotermico Dispositivo Controllo Utensili Intervenuto
"mAll_700803"	I 104.3	BOOL	// 3QM4 - MagnetotermicoVentilatore Mandrino Intervenuto
"mAll_700804"	I 104.4	BOOL	// 4QF1 - Magnetotermico Protezione trasformatore Intervenuto
"mAll_700805"	I 104.5	BOOL	// 4QF2 - Magnetotermico Protezione Utenze a 110 Vac Intervenuto
"mAll_700806"	I 104.6	BOOL	// 4QF3+4QF4 - Magnetot. Protez. Utenze 220 Vac Intervenuto
"mAll_700807"	I 104.7	BOOL	// 4QF5 - Magnetotermico Protezione Alimentazione Montronix Intervenuto
"mAll_700808"	I 105.0	BOOL	// 5QF1 - Magnetotermico Protezione Sitop 24V Uscite Intervenuto
"mAll_700809"	I 105.1	BOOL	// 5QF2 - Magnetotermico Protezione Illuminaz. Macchina Intervenuto
"mAll_700810"	I 105.2	BOOL	// 5QF3 - Magnetotermico Protezione Uscite PLC sempre alimentate Intervenuto
"mAll_700811"	I 105.3	BOOL	// 5QF4 - Magnetotermico Protezione Uscite PLC sezionate Intervenuto
"mAll_700813"	I 105.4	BOOL	// 5QF5 - Magnetotermico Protezione Alimentazione Ingressi PLC
"mAll_700814"	I 105.5	BOOL	// 5QF6 - Magnetotermico Protezione Marposs Intervenuto
"mAll_700815"	I 105.6	BOOL	// 5QF7 - Magnetotermico Protezione Elettronica CN Intervenuto
"mAll_700812"	I 105.7	BOOL	// 5QF8 - Magnetotermico Protezione Uscite Caricatore
"mAll_700816"	I 106.0	BOOL	// ERR 7280 AMT CAN.2 NON IMPOSTATI DATI
"mAll_700817"	I 106.1	BOOL	// ERR 7281 AMT CAN.2 PREALLARME
"mAll_700818"	I 106.2	BOOL	// ERR 7282 AMT CAN.2 DURATA UTENS. = 0
"mAll_700819"	I 106.3	BOOL	// ERR 7283 AMT CAN.2 CONSUM. ULTIMO UTENS.
"mAll_700820"	I 106.4	BOOL	// ERR 7284 AMT CAN.3 NON IMPOSTATI DATI
"mAll_700821"	I 106.5	BOOL	// ERR 7285 AMT CAN.3 PREALLARME
"mAll_700822"	I 106.6	BOOL	// ERR 7286 AMT CAN.3 DURATA UTENS. = 0
"mAll_700823"	I 106.7	BOOL	// ERR 7287 AMT CAN.3 CONSUM. ULTIM0 UTENS.
"mAll_700824"	I 107.0	BOOL	// ERR 7288 AMT CAN.2 PARAMETRO R SBAGLIATO
"mAll_700825"	I 107.1	BOOL	// ERR 7289 AMT CAN.3 PARAMETRO R SBAGLIATO
"mAll_700907"	I 108.7	BOOL	// ERR 7307 PL PORTE A RETE MET. N.CHIUSE
"mAll_700911"	I 109.1	BOOL	// ERR 7309 MC PORTA PARASPRUZZI N. CHIUSA
"mAll_700914"	I 109.6	BOOL	// ERR 7314 MIS. ATTESA FINCHE PRESO V.COR.
"mAll_700915"	I 109.7	BOOL	// ERR 7315 TESTA A PINZE IN POS. SCORR.
"mAll_701014"	I 113.6	BOOL	// ERR 7346 SEQ TESTA A PINZE PL A POS. 1
"mAll_701015"	I 113.7	BOOL	// ERR 7347 SEQ TESTA A PINZE PL A POS. 2
"mAll_701016"	I 114.0	BOOL	// ERR 7348 TESTA A PINZE PL IN POS.INDEF.
"mAll_701017"	I 114.1	BOOL	// ERR 7349 SEQ PL PINZA 1  CHIUDERE
"mAll_701018"	I 114.2	BOOL	// ERR 7350 SEQ PL PINZA 1  APRIRE
"mAll_701019"	I 114.3	BOOL	// ERR 7351 PL PINZA 1  IN POS. INDEF.
"mAll_701020"	I 114.4	BOOL	// ERR 7352 SEQ PL PINZA 2  CHIUDERE
"mAll_701021"	I 114.5	BOOL	// ERR 7353 SEQ PL PINZA 2  APRIRE
"mAll_701022"	I 114.6	BOOL	// ERR 7354 PL PINZA 2  IN POS. INDEF.
"mAll_701100"	I 116.0	BOOL
"mAll_701101"	I 116.1	BOOL
"mAll_701102"	I 116.2	BOOL
"mAll_701103"	I 116.3	BOOL
"mAll_701104"	I 116.4	BOOL
"mAll_701105"	I 116.5	BOOL
"mAll_701106"	I 116.6	BOOL	// ERR 7370 ARRESTO MOVIMENTO+AVANZAMENTO
"mAll_701107"	I 116.7	BOOL	// ERR 7371 COPERTA/RIBALTA  SEQ CHIUDERE
"mAll_701108"	I 117.0	BOOL	// ERR 7372 COPERTA/RIBALTA  SEQ APRIRE
"mAll_701109"	I 117.1	BOOL	// ERR 7373 COPERTA/RIBALTA  POS. INDEF.
"mAll_701110"	I 117.2	BOOL	// ERR 7374 COP./RIB.  PL IN ZONA MACC.
"mAll_701116"	I 118.0	BOOL	// ERR 7380 MM  PUNTA DESTRA SEQ RICHIAMO
"mAll_701117"	I 118.1	BOOL	// ERR 7381 MM  PUNTA DESTRA SEQ AVANZAM.
"mAll_701118"	I 118.2	BOOL	// ERR 7382 MM  PUNTA DESTRA POS. INDEF.
"mAll_701119"	I 118.3	BOOL	// ERR 7383 MM  PUNTA SIN.  SEQ RICHIAMO
"mAll_701120"	I 118.4	BOOL	// ERR 7384 MM  PUNTA SIN.  SEQ AVANZAM.
"mAll_701121"	I 118.5	BOOL	// ERR 7385 MM  PUNTA SIN.  POS. INDEF.
"mAll_701122"	I 118.6	BOOL	// ERR 7386 MM  DISP.DI CAL. SEQ. RICHIAMO
"mAll_701123"	I 118.7	BOOL	// ERR 7387 MM  DISP.DI CAL. SEQ. AVANZAM.
"mAll_701124"	I 119.0	BOOL	// ERR 7388 MM  DISP.DI CAL. POS. INDEF.
"mAll_701125"	I 119.1	BOOL	// ERR 7389 MIS. SEQ DOMANDA PEZZO SC.PART.
"mAll_701126"	I 119.2	BOOL	// ERR 7390 MIS. SEQ  V.COR.>BLOC.DATI CAN2
"mAll_701127"	I 119.3	BOOL	// ERR 7391 MIS. ATTESA  V.COR.>BL.DAT CAN2
"mAll_701128"	I 119.4	BOOL	// ERR 7392 MIS. SEQ  V.COR.>BLOC.DATI CAN3
"mAll_701129"	I 119.5	BOOL	// ERR 7393 MIS. ATTESA  V.COR.>BL.DAT CAN3
"mAll_701130"	I 119.6	BOOL	// ERR 7394 MIS. ERRORE DI CALIBRATURA
"mAll_701131"	I 119.7	BOOL	// ERR 7395 MIS. SEQ DI CALIBRATURA
"mAll_701200"	I 120.0	BOOL	// ERR 7400 MIS. MISURA DI PEZZO SCARTO
"mAll_701201"	I 120.1	BOOL	// ERR 7401 MIS. ERRORE DI MISURA
"mAll_701202"	I 120.2	BOOL	// ERR 7402 MIS. SEQ  MISURAZIONE STATICA
"mAll_701203"	I 120.3	BOOL	// ERR 7403 MIS. SEQ  MISURAIONE DINAMICA
"mAll_701204"	I 120.4	BOOL	// ERR 7404 MIS>MC  ERRORE DI PARITA
"mAll_701205"	I 120.5	BOOL	// ERR 7405 MIS>MC  ERRORE DI TRASMISSION
"mAll_701206"	I 120.6	BOOL	// ERR 7406 MIS>MC  SEQ DI TRASMISS. DATI
"mAll_701207"	I 120.7	BOOL	// ERR 7407 MIS<-MC SEQ DI TRASMISS. DATI
"mAll_701208"	I 121.0	BOOL	// ERR 7408 MIS. PROGR. DI MIS. N.TROVATO
"mAll_701209"	I 121.1	BOOL	// ERR 7409 MM  SEQ SELEZ. PROGR. DI MIS.
"mAll_701210"	I 121.2	BOOL	// ERR 7410 MM  SEQ TAVOLO -> POS.DI MIS.
"mAll_701211"	I 121.3	BOOL	// ERR 7411 MM  SEQ TAVOLO -> POS.DI CARIC.
"mAll_701212"	I 121.4	BOOL	// ERR 7412 MM  TAVOLO DI MIS. IN POS.INDEF
"mAll_701213"	I 121.5	BOOL	// ERR 7413 MM  SEQ RICHIAMO TASTATORE D
"mAll_701214"	I 121.6	BOOL	// ERR 7414 MM  SEQ ACCOSTAM. TASTATORE D
"mAll_701215"	I 121.7	BOOL	// ERR 7415 MM  TASTATORE D IN POS. INDEF.
"mAll_701216"	I 122.0	BOOL	// ERR 7416 MM  SEQ RICHIAMO TASTATORE L
"mAll_701217"	I 122.1	BOOL	// ERR 7417 MM  SEQ ACCOSTAM. TASTATORE L
"mAll_701218"	I 122.2	BOOL	// ERR 7418 MM  TASTATORE L IN POS. INDEF.
"mAll_701219"	I 122.3	BOOL	// ERR 7419 MM  SEQ  RICHIAMO STAFFA MIS.
"mAll_701220"	I 122.4	BOOL	// ERR 7420 MM  SEQ  ACCOSTAM. STAFFA MIS.
"mAll_701221"	I 122.5	BOOL	// ERR 7421 MM  STAFFA MIS. IN POS. INDEF.
"mAll_701222"	I 122.6	BOOL	// ERR 7422 MIS. QUOTA DI PEZZI SCARTI
"mAll_701223"	I 122.7	BOOL	// ERR 7423 MIS. SEQUENZA DI PEZZI SCARTI
"uNC_OK"	Q 32.0	BOOL	// KA32.0 - NC OK - Abilitazione ausiliari
"u63-9"	Q 32.1	BOOL	// KA32.1 - Abilitazione impulsi (63-9)
"u64-9"	Q 32.2	BOOL	// KA32.2 - Sblocco regolatore (64-9)
"uReset_AR_Sorvegl"	Q 32.3	BOOL	// KA32.3 - Reset modulo alimentatore e sorveglianza
"uAbil_Azion_Mandr663-9"	Q 32.4	BOOL	// KA32.4 - Abilitazione azionamento mandrino (663-9)
"uAbil_Azion_Torr_663-9"	Q 32.5	BOOL	// KA32.5 - Abilitazione azionamento assi A e B (663-9)
"uAsse_in_Oltrecorsa"	Q 32.6	BOOL	// KA32.6 - Almeno un asse è in oltrecorsa
"uAbil_Tasto_Consenso"	Q 32.7	BOOL	// KA32.7 - Abilitazione tasto di consenso
"uFreno_Mandrino"	Q 33.0	BOOL	// KA33.0 - Attivazione freno mandrino
"uLubrif_Inserita"	Q 33.1	BOOL	// KA33.1 - Lubrificazione ad impulsi inserita
"uIlluminaz_Macchina"	Q 33.2	BOOL	// KA33.2 - Attivazione illuminazione macchina
"uSblocco_Porta"	Q 33.3	BOOL	// KA33.3 - Sblocco porta paraspruzzi
"A33.4"	Q 33.4	BOOL	// KA33.4 - Disponibile
"A33.5"	Q 33.5	BOOL	// KA33.5 - Disponibile
"uSerraggio_Inserito"	Q 33.6	BOOL	// KA33.6 - 51KM2 - Sistema di serraggio inserito
"uEV_Princip_Refrig"	Q 33.7	BOOL	// KA33.7 - Attivazione EV Principale Refrigerante
"uLavaggio_Carrello"	Q 34.0	BOOL	// KA34.0 - Lavaggio carrello inferiore
"uMarposs_Trend"	Q 34.1	BOOL	// KA34.1 - Marposs - Valore trend di misura
"uMarposs_Rich_Dati"	Q 34.2	BOOL	// KA34.2 - Marposs - Richiesta nuovi dati
"uMarposs_Reset_Trend"	Q 34.3	BOOL	// KA34.3 - Marposs - Reset Trend
"uCanc_All_Olio"	Q 34.4	BOOL	// KA34.4 - Controllo livello olio cancellazione allarme
"uColonna_Verde"	Q 34.5	BOOL	// KA34.5 - 50HL3 - Colonna luminosa elemento verde
"uColonna_Arancio"	Q 34.6	BOOL	// KA34.6 - 50HL4 - Colonna luminosa elemento arancio
"uColonna_Rosso"	Q 34.7	BOOL	// KA34.7 - 50HL5 - Colonna luminosa elemento rosso
"uCil_Serrag_Avanti"	Q 35.0	BOOL	// KA35.0 - 52YV4A - Cilindro di serraggio avanti
"uCil_Serrag_Indietro"	Q 35.1	BOOL	// KA35.1 - 52YV4B - Cilindro di serraggio ritorno
"uCannotto_Avanti"	Q 35.2	BOOL	// KA35.2 - 52YV5A - Cannotto di contropunta avanti
"uCannotto_Indietro"	Q 35.3	BOOL	// KA35.3 - 52YV5B - Cannotto di contropunta ritorno
"uSbloccag_Controp"	Q 35.4	BOOL	// KA35.4 - 52YV6 - Sblocaggio Contropunta
"uSblocco_Freno_X1"	Q 35.5	BOOL	// KA35.5 - Sblocco Freno Asse X1
"uSblocco_Freno_X2"	Q 35.6	BOOL	// KA35.6 - Sblocco Freno Asse X2
"uMonitor_Impulso_Ciclo"	Q 35.7	BOOL	// KA35.7 - Monitor di Manutenzione - Impulso ciclo
"uDisser_Utens_Blocco_A1"	Q 36.0	BOOL	// KA36.0 - 53YV1 - Disserrare utensili blocco sistema A
"uDisser_Utens_Blocco_A2"	Q 36.1	BOOL	// KA36.1 - 53YV2 - Disserrare utensili blocco sistema A
"uDisser_Utens_Blocco_B1"	Q 36.2	BOOL	// KA36.2 - 53YV3 - Disserrare utensili blocco sistema B
"uDisser_Utens_Blocco_B2"	Q 36.3	BOOL	// KA36.3 - 53YV4 - Disserrare utensili blocco sistema B
"uTorretta_A_Bloccaggio"	Q 36.4	BOOL	// KA36.4 - 53YV5A - Torretta A Bloccaggio
"uTorretta_A_Sbloccaggio"	Q 36.5	BOOL	// KA36.5 - 53YV5B - Torretta A Sbloccaggio
"uTorretta_B_Bloccaggio"	Q 36.6	BOOL	// KA36.6 - 53YV6A - Torretta B Bloccaggio
"uTorretta_B_Sbloccaggio"	Q 36.7	BOOL	// KA36.7 - 53YV6B - Torretta B Sbloccaggio
"uRiparo_Scorr_Apertura"	Q 37.0	BOOL	// KA37.0 - 54YV4A - Riparo scorrevole apertura
"uRiparo_Scorr_Chiusura"	Q 37.1	BOOL	// KA37.1 - 54YV4B - Riparo scorrevole chiusura
"A37.2"	Q 37.2	BOOL
"uRenishaw_in_misura"	Q 37.3	BOOL	// KA37.3 - 51KM3 - Braccio Renishaw in posiz. di misura
"uRenishaw_a_riposo"	Q 37.4	BOOL	// KA37.4 - 51KM4 - Braccio Renishaw a riposo
"uRiparo_Renishaw_Chiuso"	Q 37.5	BOOL	// KA37.5 - 54YV1A - Riparo Renishaw chiuso
"uRiparo_Renishaw_Aperto"	Q 37.6	BOOL	// KA37.6 - 54YV1B - Riparo Renishaw aperto
"uFreno_Renishaw_Chiuso"	Q 37.7	BOOL	// KA37.7 - Braccio Renishaw Freno inserito
"uMDE_Macch_in_Auto"	Q 38.0	BOOL	// REG.DATI MC  MACCH. IN CICLO AUTOM.
"uMDE_Arresto_Anomalia"	Q 38.1	BOOL	// REG.DATI MC  ARRESTO MACCH. (ANOMALIA)
"uMDE_Arresto_Carico"	Q 38.2	BOOL	// REG.DATI MC  ARRESTO MACCH. (CARICO)
"uMDE_Arresto_Scarico"	Q 38.3	BOOL	// REG.DATI MC  ARRESTO MACCH. (SCARICO)
"uMDE_Arresto_CU"	Q 38.4	BOOL	// REG.DATI MC  ARRESTO MACCH. (Cambio Utensile programmato)
"uMDE_Arresto_Tipo_Pezzo"	Q 38.5	BOOL	// REG.DATI MC  ARRESTO MACCH. (TIPO PEZZO)
"uMDE_Arresto_Incerto"	Q 38.6	BOOL	// REG.DATI MC  ARRESTO MACCH. (INCERTO)
"uMDE_Macch_Funziona"	Q 38.7	BOOL	// REG.DATI MC  MACCHINA FUNZIONA
"uMDE_Imp_Cont_Pz_Finiti"	Q 39.0	BOOL	// REG.DATI MC  IMPULSO Conteggio Pezzi Finiti
"uMDE_Imp_Pz_Scarto"	Q 39.1	BOOL	// REG.DATI MC  IMPULSO DI PEZZO SCARTO
"uMDE_Tipo_Pz_Bit1"	Q 39.2	BOOL	// REG.DATI MC  TIPO PEZZO  BIT 1
"uMDE_Tipo_Pz_Bit2"	Q 39.3	BOOL	// REG.DATI MC  TIPO PEZZO  BIT 2
"uMDE_Tipo_Pz_Bit3"	Q 39.4	BOOL	// REG.DATI MC  TIPO PEZZO  BIT 3
"uMDE_Tipo_Pz_Bit4"	Q 39.5	BOOL	// REG.DATI MC  TIPO PEZZO  BIT 4
"uMDE_Tipo_Pz_Parità"	Q 39.6	BOOL	// REG.DATI MC  TIPO PEZZO  PARITA
"uMDE_Riserva"	Q 39.7	BOOL	// REG.DATI MC  RISERVA
"uMontr_A_Nuovo_Pz"	Q 40.0	BOOL	// GF->MONTRONIX SIS-A  NUOVO PEZZO
"uMontr_A_Nuovo_Utens"	Q 40.1	BOOL	// GF->MONTRONIX SIS-A  NUOVO UTENSILE
"uMontr_A_Cancel_Allarme"	Q 40.2	BOOL	// GF->MONTRONIX SIS-A  CANCELL. L'ALLARME
"uMontr_A_Amplificat_Ins"	Q 40.3	BOOL	// GF->MONTRONIX SIS-A  AMPLIFICATORE INS
"uMontr_A_Selez_Pz/Utens"	Q 40.4	BOOL	// GF->MONTRONIX SIS-A  SELEZ. PEZZO/UTENS.
"uMontr_A_Ris"	Q 40.5	BOOL	// GF->MONTRONIX SIS-A  RISERVA
"uMontr_A_Nel_Ciclo"	Q 40.6	BOOL	// GF->MONTRONIX SIS-A  NEL CICLO
"uMontr_A_Ricon_Rapido"	Q 40.7	BOOL	// GF->MONTRONIX SIS-A  RICONOSC.DEL RAPIDO
"uMontr_A_Dati_Bit1"	Q 41.0	BOOL	// GF->MONTRONIX SIS-A  DATI  BIT 1
"uMontr_A_Dati_Bit2"	Q 41.1	BOOL	// GF->MONTRONIX SIS-A  DATI  BIT 2
"uMontr_A_Dati_Bit4"	Q 41.2	BOOL	// GF->MONTRONIX SIS-A  DATI  BIT 4
"uMontr_A_Dati_Bit8"	Q 41.3	BOOL	// GF->MONTRONIX SIS-A  DATI  BIT 8
"uMontr_A_Dati_Bit16"	Q 41.4	BOOL	// GF->MONTRONIX SIS-A  DATI  BIT 16
"uMontr_A_Dati_Bit32"	Q 41.5	BOOL	// GF->MONTRONIX SIS-A  DATI  BIT 32
"uMontr_A_Disp1"	Q 41.6	BOOL	// GF->MONTRONIX SIS-A Disponibile
"uMontr_A_Disp2"	Q 41.7	BOOL	// GF->MONTRONIX SIS-A Disponibile
"uMontr_B_Nuovo_Pz"	Q 42.0	BOOL	// GF->MONTRONIX SIS-B  NUOVO PEZZO
"uMontr_B_Nuovo_Utens"	Q 42.1	BOOL	// GF->MONTRONIX SIS-B  NUOVO UTENSILE
"uMontr_B_Cancel_Allarme"	Q 42.2	BOOL	// GF->MONTRONIX SIS-B  CANCELL. L'ALLARME
"uMontr_B_Amplificat_Ins"	Q 42.3	BOOL	// GF->MONTRONIX SIS-B  AMPLIFICATORE INS
"uMontr_B_Selez_Pz/Utens"	Q 42.4	BOOL	// GF->MONTRONIX SIS-B  SELEZ. PEZZO/UTENS.
"uMontr_B_Ris"	Q 42.5	BOOL	// GF->MONTRONIX SIS-B  RISERVA
"uMontr_B_Nel_Ciclo"	Q 42.6	BOOL	// GF->MONTRONIX SIS-B  NEL CICLO
"uMontr_B_Ricon_Rapido"	Q 42.7	BOOL	// GF->MONTRONIX SIS-B  RICONOSC.DEL RAPIDO
"uMontr_B_Dati_Bit1"	Q 43.0	BOOL	// GF->MONTRONIX SIS-B  DATI  BIT 1
"uMontr_B_Dati_Bit2"	Q 43.1	BOOL	// GF->MONTRONIX SIS-B  DATI  BIT 2
"uMontr_B_Dati_Bit4"	Q 43.2	BOOL	// GF->MONTRONIX SIS-B  DATI  BIT 4
"uMontr_B_Dati_Bit8"	Q 43.3	BOOL	// GF->MONTRONIX SIS-B  DATI  BIT 8
"uMontr_B_Dati_Bit16"	Q 43.4	BOOL	// GF->MONTRONIX SIS-B  DATI  BIT 16
"uMontr_B_Dati_Bit32"	Q 43.5	BOOL	// GF->MONTRONIX SIS-B  DATI  BIT 32
"uMontr_B_Disp1"	Q 43.6	BOOL	// GF->MONTRONIX SIS-B Disponibile
"uMontr_B_Disp2"	Q 43.7	BOOL	// GF->MONTRONIX SIS-B Disponibile
"uPL_Aux_ON"	Q 44.0	BOOL	// GF->PL  Ausiliari inseriti
"uPL_Ciclo_Auto"	Q 44.1	BOOL	// GF->PL  Ciclo Automatico in corso
"uPL_Portare_Pezzo"	Q 44.2	BOOL	// GF->PL  SEGNALE PRELIM.  PORTARE PEZZO
"uPL_Consenso_Prelievo"	Q 44.3	BOOL	// GF->PL  Consenso al ciclo di prelievo
"uPL_Consenso_Attesa"	Q 44.4	BOOL	// GF->PL  Consenso posizione di attesa
"uPL_Consenso_Deposito"	Q 44.5	BOOL	// GF->PL  Consenso al ciclo di deposito
"uPL_Pezzo_Sbloccato"	Q 44.6	BOOL	// GF->PL  Pezzo Sbloccato
"uPL_Ciclo_Cambio_Pezzo"	Q 44.7	BOOL	// GF->PL  Ciclo speciale cambio pezzo
"uPL_Pezzo_Bloccato"	Q 45.0	BOOL	// GF->PL  Pezzo Bloccato
"uPL_Porta_Pezzo"	Q 45.1	BOOL	// GF->PL  Porta Pezzo (tipo pezzo OK)
"uPL_Svuotam_Macch"	Q 45.2	BOOL	// GF->PL  Svuotamento macchina
"uPL_Pezzo_Prebloccato"	Q 45.3	BOOL	// GF->PL  Pezzo Prebloccato
"uPL_Macch_Senza_Pezzo"	Q 45.4	BOOL	// GF->PL  Macchina Senza Pezzo
"uPL_Pezzo_Finito"	Q 45.5	BOOL	// GF->PL  Pezzo Finito in Macchina
"uPL_Disp1"	Q 45.6	BOOL	// GF->PL  Disponibile
"uPL_Disp2"	Q 45.7	BOOL	// GF->PL  Disponibile
"uPM_PEZZO_FISSATO"	Q 64.0	BOOL	// QUADRO DI COM.MC  PEZZO FISSATO
"uPM_ARRESTO_FINE_CICLO"	Q 64.3	BOOL	// QUADRO COM.MC  ARRESTO ALLA FINE CICLO
"uPM_SBLOCCAGGIO_PORTA"	Q 65.1	BOOL	// QUADRO DI COM.MC  SBLOCCAGGIO PORTA
"mBL_Can1_Coordin_Canali"	Q 68.0	BOOL	// BLOCCO LETT. CAN.1 COORDINAM. CANALI
"mBL_Can1_Param_R99=1"	Q 68.1	BOOL	// BLOCCO LETT. CAN.1 PARAMETRO R 99=1
"mBL_Can1_Param_R99=0"	Q 68.2	BOOL	// BLOCCO LETT. CAN.1 PARAMETRO R 99=0
"mBL_Can1_Contr_Progr"	Q 68.3	BOOL	// BLOCCO LETT. CAN.1 CONTROLLO PROGRAMMI
"mBL_Can1_ImposDatiFond"	Q 68.4	BOOL	// BLOCCO LETT. CAN.1 IMPOSTAZ. DATI FOND.
"mBL_Can1_Lettura_R100"	Q 68.5	BOOL	// BLOCCO LETT. CAN.1 LETTURA DI R100
"mBL_Can1_Mediante_M868"	Q 68.6	BOOL	// BLOCCO LETT. CAN.1 MEDIANTE M868
"mBL_Can1_Sincronizzaz"	Q 69.0	BOOL	// BLOCCO LETT. CAN.1 SINCRONIZZAZ. CAN.1
"mBL_Can1_Err_SINCRON"	Q 69.1	BOOL	// BLOCCO LETT. CAN.1 ERR 7211 DI SINCRON.
"mBL_Can1_MISURAZ"	Q 69.2	BOOL	// BLOCCO LETT. CAN.1 MISURAZ. PEZZI
"mBL_Can1_GENERALITA"	Q 69.3	BOOL	// BLOCCO LETT. CAN.1 GENERALITA
"mBL_Can1_LIBERAZIONE"	Q 69.4	BOOL	// BLOCCO LETT. CAN.1 LIBERAZIONE AUTOM.
"mBL_Can1_SELEZIONE_TIPO"	Q 69.5	BOOL	// BLOCCO LETT. CAN.1 SELEZIONE TIPO PEZZO
"mBL_Can1_AIUTO_LETTURA"	Q 69.6	BOOL	// BLOCCO LETT. CAN.1 AIUTO LETTURA PARAM.R
"mBL_Can1_AVVIO/RIC.OR"	Q 69.7	BOOL	// BL.LETT. CAN.1 LOGICA AVVIO/RIC.ORIG.AUT
"mStop_Ciclo_Can1_GENE"	Q 70.0	BOOL	// BLOC.CICLO CAN.1 GENERALITA (PB80)
"mStopCicloCan1_ContaPezz"	Q 70.1	BOOL	// BLOC.CICLO CAN.1 CONTATORE PEZZI
"mStop_Ciclo_Can1_DURAT"	Q 70.2	BOOL	// BLOC.CICLO CAN.1 DURATA CICLO SUPERATA
"mStop_Ciclo_Can1_Richies"	Q 70.7	BOOL	// BLOC.CICLO CAN.1 RICHIESTE DEL CLIENTE
"mBL_Can2_Arresto_Emerg"	Q 71.0	BOOL	// BLOC.LETT. CAN.2 ARRESTO DI EMERGENZA
"mBL_Can2_MANDRINO"	Q 71.1	BOOL	// BLOC.LETT. CAN.2 MANDRINO 1
"mBL_Can2_DISP_DI_SER"	Q 71.3	BOOL	// BLOC.LETT. CAN.2 DISP. DI SERRAGGIO
"mBL_Can2_SIST_DI_REF"	Q 71.4	BOOL	// BLOC.LETT. CAN.2 SIST. DI REFRIGERANTE
"mBL_Can2_TORRETTA_1"	Q 71.5	BOOL	// BLOC.LETT. CAN.2 TORRETTA 1
"mBL_Can2_CONTROT"	Q 71.6	BOOL	// BLOC.LETT. CAN.2 CONTROTESTA A CN
"mBL_Can2_COPERTA/R"	Q 71.7	BOOL	// BLOC.LETT. CAN.2 COPERTA/RIBALTA
"mBL_Can2_LUNETTA"	Q 72.0	BOOL	// BLOC.LETT. CAN.2 LUNETTA
"mBL_Can2_DISP_DI_MIS"	Q 72.3	BOOL	// BLOC.LETT. CAN.2 DISP. DI MISURA UTENS.
"mBL_Can2_ROTTURA_U"	Q 72.4	BOOL	// BLOC.LETT. CAN.2 ROTTURA UTENSILE
"mBL_Can2_MOTORI_DI"	Q 72.5	BOOL	// BLOC.LETT. CAN.2 MOTORI DI AVANZAMENTO
"mBL_Can2_Param_R99=1"	Q 72.6	BOOL	// BLOC.LETT. CAN.2 PARAMETRI R 99=1
"mBL_Can2_Param_R99=0"	Q 72.7	BOOL	// BLOC.LETT. CAN.2 PARAMETRI R 99=0
"mBL_Can2_Sincronizzaz"	Q 73.0	BOOL	// BLOC.LETT. CAN.2 SINCRONIAZZAZIONE
"mBL_Can2_ERR_7212_SINCRO"	Q 73.1	BOOL	// BLOC.LETT. CAN.2 ERR 7212 SINCRONIZZ.
"mBL_Can2_CONTR_PROGRA"	Q 73.3	BOOL	// BLOC.LETT. CAN.2 CONTR. PROGRAMMI
"mBL_Can2_PORTA_PAR"	Q 73.4	BOOL	// BLOC.LETT. CAN.2 PORTA PARASPRUZZI AUTOM
"mBL_Can2_COMMUT_RA"	Q 73.6	BOOL	// BLOC.LETT. CAN.2 COMMUT. RAGGIO/DIAMETRO
"mBL_Can2_AGGIUNGERE"	Q 73.7	BOOL	// BLOC.LETT. CAN.2 AGGIUNGERE POS. ASSIALE
"mBL_Can2_Mis_TrasmValCor"	Q 74.0	BOOL	// BLOC.LETT. CAN.2 MIS. TRASMISS. VAL.CORR
"mBL_Can2_Misuraz_Pezzi"	Q 74.2	BOOL	// BLOC.LETT. CAN.2 MISURAZIONE PEZZI
"mBL_Can2_CALIBRATURA_UT"	Q 74.3	BOOL	// BLOC.LETT. CAN.2 CALIBRATURA UTENSILI
"mBL_Can2_AMT_D_R101-R112"	Q 74.4	BOOL	// BLOC.LETT. CAN.2 AMT  NO.D IN R101-R112
"mBL_Can2_AMT_LETTURA"	Q 74.5	BOOL	// BLOC.LETT. CAN.2 AMT  LETTURA PARAM. R
"mBL_Can2_AMT  ERRORI"	Q 74.6	BOOL	// BLOC.LETT. CAN.2 AMT  ERRORI
"mBL_Can2_da_AB75_a_AB80"	Q 74.7	BOOL	// BLOC.LETT. CAN.2 DA AB75 A AB80
"mBL_Can2_Misuraz_Pezzi?"	Q 75.2	BOOL	// BLOC.LETT. CAN.2 MISURAZIONE PEZZI
"mBL_Can2_BLOCC. PORTA"	Q 75.3	BOOL	// BLOC.LETT. CAN.2 BLOCC. PORTA PARASPRUZZ
"mBL_Can2_RICERCA ORIG"	Q 75.7	BOOL	// BLOC.LETT. CAN.2 RICERCA ORIGINE INTELL.
"mBL_Can2_INTERR_ROTAZ"	Q 76.7	BOOL	// BLOC.LETT. CAN.2 INTERR. DI ROTAZIONE
"mBL_Can2_LIBERAZIONE AUT"	Q 78.0	BOOL	// BLOC.LETT. CAN.2 LIBERAZIONE AUTOMATICA
"mBL_Can2_GENERALITA"	Q 79.3	BOOL	// BLOC.LETT. CAN.2 GENERALITA
"mBL_Can3_Arresto_Emerg"	Q 81.0	BOOL	// BLOC.LETT. CAN.3 ARRESTO DI EMERGENZA
"mBL_Can3_MANDRINO 1"	Q 81.1	BOOL	// BLOC.LETT. CAN.3 MANDRINO 1
"mBL_Can3_DISP. DI SERRA"	Q 81.3	BOOL	// BLOC.LETT. CAN.3 DISP. DI SERRAGGIO
"mBL_Can3_SIST. REFRIGER"	Q 81.4	BOOL	// BLOC.LETT. CAN.3 SIST. REFRIGERANTE
"mBL_Can3_TORRETTA 2"	Q 81.5	BOOL	// BLOC.LETT. CAN.3 TORRETTA 2
"mBL_Can3_CONTROTESTA A"	Q 81.6	BOOL	// BLOC.LETT. CAN.3 CONTROTESTA A CN
"mBL_Can3_COPERTA/RIBA"	Q 81.7	BOOL	// BLOC.LETT. CAN.3 COPERTA/RIBALTA
"mBL_Can3_LUNETTA"	Q 82.0	BOOL	// BLOC.LETT. CAN.3 LUNETTA
"mBL_Can3_DISP_DI MIS_UT"	Q 82.3	BOOL	// BLOC.LETT. CAN.3 DISP. DI MIS. UTENS.
"mBL_Can3_ROTTURA UTENS"	Q 82.4	BOOL	// BLOC.LETT. CAN.3 ROTTURA UTENSILE
"mBL_Can3_Param_R99=1"	Q 82.6	BOOL	// BLOC.LETT. CAN.3 PARAMETRI R 99=1
"mBL_Can3_Param_R99=0"	Q 82.7	BOOL	// BLOC.LETT. CAN.3 PARAMETRI R 99=0
"mBL_Can3_Sincronizzaz"	Q 83.0	BOOL	// BLOC.LETT. CAN.3 SINCRONIZZAZIONE CAN.3
"mBL_Can3_ERRORE 7213"	Q 83.1	BOOL	// BLOC.LETT. CAN.3 ERRORE 7213
"mBL_Can3_CONTROLLO"	Q 83.3	BOOL	// BLOC.LETT. CAN.3 CONTROLLO PROGRAMMI
"mBL_Can3_PORTA PARASP"	Q 83.4	BOOL	// BLOC.LETT. CAN.3 PORTA PARASPRUZZI AUTOM
"mBL_Can3_AGGIUNGERE"	Q 83.7	BOOL	// BLOC.LETT. CAN.3 AGGIUNGERE POS. ASSIALE
"mBL_Can3_Mis_TrasmValCor"	Q 84.0	BOOL	// BLOC.LETT. CAN.3 MIS. TRASMISS. VAL.CORR
"mBL_Can3_MISURAZIONE"	Q 84.2	BOOL	// BLOC.LETT. CAN.3 MISURAZIONE PEZZI
"mBL_Can3_CALIBRATURA"	Q 84.3	BOOL	// BLOC.LETT. CAN.3 CALIBRATURA UTENSILI
"mBL_Can3_AMT_D_R101-R112"	Q 84.4	BOOL	// BLOC.LETT. CAN.3 AMT  NO. D IN R101-R112
"mBL_Can3_AMT  LETTURA"	Q 84.5	BOOL	// BLOC.LETT. CAN.3 AMT  LETTURA PARAM. R
"mBL_Can3_AMT  ERRORI"	Q 84.6	BOOL	// BLOC.LETT. CAN.3 AMT  ERRORI
"mBL_Can3_DA AB85 A AB90"	Q 84.7	BOOL	// BLOC.LETT. CAN.3 DA AB85 A AB90
"mBL_Can3_BLOCC. PORTA"	Q 85.3	BOOL	// BLOC.LETT. CAN.3 BLOCC. PORTA PARASPRUZ.
"mBL_Can3_RICERCA ORIGI"	Q 85.7	BOOL	// BLOC.LETT. CAN.3 RICERCA ORIGINE INTELL.
"mBL_Can3_INTERR. DI ROT"	Q 86.7	BOOL	// BLOC.LETT. CAN.3 INTERR. DI ROTAZIONE
"mBL_Can3_LIBERAZIONE"	Q 88.0	BOOL	// BLOC.LETT. CAN.3 LIBERAZIONE AUTOMATICA
"mBL_Can3_GENERALITA"	Q 89.3	BOOL	// BLOC.LETT. CAN.3 GENERALITA
"mArr_Emerg_CAN2+3_Cdo_Av"	Q 91.0	BOOL	// ARR.DI EM. CAN.2+3 COM.AVANZ. MACCH.
"ARR.DI EM. CAN.2+3 DISP."	Q 91.1	BOOL	// ARR.DI EM. CAN.2+3 DISP. DI SERRAGGIOA
"ARR.DI EM. CAN.2+3 MAN"	Q 91.2	BOOL	// ARR.DI EM. CAN.2+3 MANDRINO 1
"mArrestoEmerCan2+3xTorr1"	Q 91.3	BOOL	// ARR.DI EM. CAN.2+3 TORRETTA 1
"mArrestoEmerCan2+3xTorr2"	Q 91.4	BOOL	// ARR.DI EM. CAN.2+3 TORRETTA 2
"ARR.DI EM. CAN.2+3 RILEV"	Q 91.7	BOOL	// ARR.DI EM. CAN.2+3 RILEV.GEN. DI ERRORI
"ARR.DI EM. CAN.2+3 LUNE"	Q 92.0	BOOL	// ARR.DI EM. CAN.2+3 LUNETTA
"mStopAv_Can2+3_ContrProg"	Q 93.1	BOOL	// ARR.MOVIM. CAN.2+3 CONTR. PROGRAMMI
"mStopAv_Can2+3 CON"	Q 93.2	BOOL	// ARR.MOVIM. CAN.2+3 CONTR. PROGRAMMI
"mStopAv_Can2+3 ERR"	Q 97.0	BOOL	// ARR.AVANZ. CAN.2+3 ERR7070/7071
"mStopAv_Can2+3_ComAvMac"	Q 97.1	BOOL	// ARR.AVANZ. CAN.2+3 COM.AVANZAM. MACCH.
"mStopAv_Can2+3 MAN"	Q 97.2	BOOL	// ARR.AVANZ. CAN.2+3 MANDRINO 1
"mStopAv_Can2+3 ROTT"	Q 97.4	BOOL	// ARR.AVANZ. CAN.2+3 ROTTURA UTENSILE
"mStopAv_Can2+3_Com_Avan"	Q 97.6	BOOL	// ARR.AVANZ. CAN.2+3 COMANDO AVANZAMENTO
"mStopAv_Can2+3 M704"	Q 98.5	BOOL	// ARR.AVANZ. CAN.2+3 M704 CANALE 2
"mStopAv_Can2+3 M70"	Q 98.6	BOOL	// ARR.AVANZ. CAN.2+3 M704 CANALE 3
"mStopAv_Can2+3 ARRE"	Q 98.7	BOOL	// ARR.AVANZ. CAN.2+3 ARRESTO MANDRINO
"mStopMandr_CAN.2+3 ERR70"	Q 99.0	BOOL	// INTER.ROT. CAN.2+3 ERR7070/7071
"mINTER.ROT. CAN.2+3 MAN"	Q 99.2	BOOL	// INTER.ROT. CAN.2+3 MANDRINO 1
"mINTER.ROT. CAN.2+3 ROTT"	Q 99.4	BOOL	// INTER.ROT. CAN.2+3 ROTTURA UTENSILE
"mStop_Ciclo_Can2+3 RILEV"	Q 101.1	BOOL	// BLOC.CICLO CAN.2+3 RILEV.GEN. DI ERRORI
"mStop_Ciclo_Can2+3 MAN"	Q 101.2	BOOL	// BLOC.CICLO CAN.2+3 MANDRINO 1
"mStopCiclo_Can2+3_xLubr"	Q 101.3	BOOL	// BLOC.CICLO CAN.2+3 LUBRIFIC. AD IMPULSI
"mStop_Ciclo_Can2+3 POMP"	Q 101.4	BOOL	// BLOC.CICLO CAN.2+3 POMPA AD ALTA PRESS.
"mStop_Ciclo_Can2+3 ROTT"	Q 101.7	BOOL	// BLOC.CICLO CAN.2+3 ROTTURA UTENSILE
"mStop_Ciclo_Can2+3 TRAS"	Q 102.3	BOOL	// BLOC.CICLO CAN.2+3 TRASPORTATRUCIOLI
"mStopCicloCan2+3_MisScar"	Q 102.4	BOOL	// BLOC.CICLO CAN.2+3 MIS. SEQU.PEZZI SCARTI
"mStop_Ciclo_Can2+3 MIS."	Q 102.5	BOOL	// BLOC.CICLO CAN.2+3 MIS. QUOTA PEZZI SCAR
"mStop_Ciclo_Can2+3 AMT"	Q 102.6	BOOL	// BLOC.CICLO CAN.2+3 AMT ANOMALIA
"mStop_Ciclo_Can2+3"	Q 102.7	BOOL	// BLOC.CICLO CAN.2+3
"mBL_Can4_Arresto_Emerg"	Q 103.0	BOOL	// BLOC.LETT. CAN.4  ARRESTO DI EMERGENZA
"mBL_Can4  MANDRINO 1"	Q 103.1	BOOL	// BLOC.LETT. CAN.4  MANDRINO 1
"mBL_Can4  DISP. DI SERR"	Q 103.3	BOOL	// BLOC.LETT. CAN.4  DISP. DI SERRAGGIO
"mBL_Can4  REFRIGERANTE"	Q 103.4	BOOL	// BLOC.LETT. CAN.4  REFRIGERANTE
"mBL_Can4  CONTROTESTA"	Q 103.5	BOOL	// BLOC.LETT. CAN.4  CONTROTESTA A CN
"mBL_Can4  COPERTA/RIBA"	Q 104.0	BOOL	// BLOC.LETT. CAN.4  COPERTA/RIBALTA
"mBL_Can4  DISP_MIS_UT"	Q 104.1	BOOL	// BLOC.LETT. CAN.4  DISP.DI MIS. UTENSILI
"mBL_Can4  LUNETTA"	Q 104.7	BOOL	// BLOC.LETT. CAN.4  LUNETTA
"mBL_Can4_Sincronizzaz"	Q 105.0	BOOL	// BLOC.LETT. CAN.4  SINCRONIZZAZIONE CAN.4
"mBL_Can4  ERRORE 7214"	Q 105.1	BOOL	// BLOC.LETT. CAN.4  ERRORE 7214
"mBL_Can4  CONTR. PROG"	Q 105.3	BOOL	// BLOC.LETT. CAN.4  CONTR. PROGRAMMI
"mBL_Can4  MAC. DI MISU"	Q 105.4	BOOL	// BLOC.LETT. CAN.4  MAC. DI MISURA 1
"mBL_Can4  MIS.  SCARTO"	Q 105.6	BOOL	// BLOC.LETT. CAN.4  MIS.  SCARTO PARTICOL.
"mBL_Can4  AGGIUNGERE"	Q 105.7	BOOL	// BLOC.LETT. CAN.4  AGGIUNGERE POS. ASSIAL
"mBL_Can4_Param_R99=1"	Q 106.0	BOOL	// BLOC.LETT. CAN.4  PARAMETRI R99=1
"mBL_Can4_Param_R99=0"	Q 106.1	BOOL	// BLOC.LETT. CAN.4  PARAMETRI R99=0
"mBL_Can4  SVOLGIM. DI"	Q 106.2	BOOL	// BLOC.LETT. CAN.4  SVOLGIM. DI MISURAZ.
"mBL_Can4  PROGR. DI MI"	Q 106.3	BOOL	// BLOC.LETT. CAN.4  PROGR. DI MISURA A
"mBL_Can4_da_AB107aAB112"	Q 106.7	BOOL	// BLOC.LETT. CAN.4  DA AB107 A AB112
"mBL_Can4  INTERR. DI RO"	Q 107.7	BOOL	// BLOC.LETT. CAN.4  INTERR. DI ROTAZIONE
"mBL_Can4"	Q 108.7	BOOL	// BLOC.LETT. CAN.4
"mBL_Can4_Generalita'"	Q 109.3	BOOL	// BLOC.LETT. CAN.4  GENERALITA
"NOTAUS  KNL4 SPDL1"	Q 114.2	BOOL	// NOTAUS  KNL4 SPDL1
"mStop_Avanz_CAN.4  ERR7"	Q 116.0	BOOL	// ARR.MOVIM. CAN.4  ERR7370
"mStop_Avanz_CAN.4  RILEV"	Q 116.1	BOOL	// ARR.MOVIM. CAN.4  RILEVAM. GEN.DI ERRORI
"mStop_Avanz_CAN.4  CON"	Q 116.3	BOOL	// ARR.MOVIM. CAN.4  CONTR. PROGRAMMI
"COM.AVANZ. CAN.4  RILE"	Q 120.2	BOOL	// COM.AVANZ. CAN.4  RILEVAM. GEN.DI ERRORI
"mStopAvan_Can4xStopMandr"	Q 120.7	BOOL	// COM.AVANZ. CAN.4  INTERR. DI ROTAZIONE
"COM.AVANZ. CAN.4  MAN"	Q 121.2	BOOL	// COM.AVANZ. CAN.4  MANDRINO 1
"ALARM_SQ"	SFC 17	SFC 17	// Generate Block-Related Messages with Acknowledgment
"TIME_TCK"	SFC 64	SFC 64	// Read the System Time
END_SYMBOL_TABLE

TYPE UDT 2
VERSION : 0.0
  STRUCT
   C1 : STRUCT 	//From Channel 1
    FDD_5100xx : ARRAY  [0 .. 15 ] OF //Feed disable A.no.51000-510015
    BOOL ;
    FDD_RID_5101xx : ARRAY  [0 .. 31 ] OF //Feed and read-in disable A.no.510100-510131
    BOOL ;
    RID_5102xx : ARRAY  [0 .. 31 ] OF //Read-in disable A.no.510200-510231
    BOOL ;
    NCSD_5103xx : ARRAY  [0 .. 15 ] OF //NC start disable A.no.510300-510315
    BOOL ;
    FdStop_1_5111xx : ARRAY  [0 .. 15 ] OF //Feed stop GEOaxis 1 A.no.511100-511115
    BOOL ;
    FdStop_2_5112xx : ARRAY  [0 .. 15 ] OF //Feed stop GEOaxis 2 A.no.511200-511215
    BOOL ;
    FdStop_3_5113xx : ARRAY  [0 .. 15 ] OF //Feed stop GEOaxis 3 A.no.511300-511315
    BOOL ;
   END_STRUCT ;
   C2 : STRUCT 	//From Channel 2
    FDD_5200xx : ARRAY  [0 .. 15 ] OF //Feed disable A.no.520000-520015
    BOOL ;
    FDD_RID_5201xx : ARRAY  [0 .. 31 ] OF //Feed and read-in disable A.no.520100-520131
    BOOL ;
    RID_5202xx : ARRAY  [0 .. 31 ] OF //Read-in disable A.no.520200-520231
    BOOL ;
    NCSD_5203xx : ARRAY  [0 .. 15 ] OF //NC start disable A.no.520300-520315
    BOOL ;
    FdStop_1_5211xx : ARRAY  [0 .. 15 ] OF //Feed stop GEOaxis 1 A.no.521100-521115
    BOOL ;
    FdStop_2_5212xx : ARRAY  [0 .. 15 ] OF //Feed stop GEOaxis 2 A.no.521200-521215
    BOOL ;
    FdStop_3_5213xx : ARRAY  [0 .. 15 ] OF //Feed stop GEOaxis 3 A.no.521300-521315
    BOOL ;
   END_STRUCT ;
   C3 : STRUCT 	//From Channel 3
    FDD_5300xx : ARRAY  [0 .. 15 ] OF //Feed disable A.no.530000-530015
    BOOL ;
    FDD_RID_5301xx : ARRAY  [0 .. 31 ] OF //Feed and read-in disable A.no.530100-530131
    BOOL ;
    RID_5302xx : ARRAY  [0 .. 31 ] OF //Read-in disable A.no.530200-530231
    BOOL ;
    NCSD_5303xx : ARRAY  [0 .. 15 ] OF //NC start disable A.no.530300-530315
    BOOL ;
    FdStop_1_5311xx : ARRAY  [0 .. 15 ] OF //Feed stop GEOaxis 1 A.no.531100-531115
    BOOL ;
    FdStop_2_5312xx : ARRAY  [0 .. 15 ] OF //Feed stop GEOaxis 2 A.no.531200-531215
    BOOL ;
    FdStop_3_5313xx : ARRAY  [0 .. 15 ] OF //Feed stop GEOaxis 3 A.no.531300-531315
    BOOL ;
   END_STRUCT ;
   C4 : STRUCT 	//From Channel 4
    FDD_5400xx : ARRAY  [0 .. 15 ] OF //Feed disable A.no.540000-540015
    BOOL ;
    FDD_RID_5401xx : ARRAY  [0 .. 31 ] OF //Feed and read-in disable A.no.540100-540131
    BOOL ;
    RID_5402xx : ARRAY  [0 .. 31 ] OF //Read-in disable A.no.540200-540231
    BOOL ;
    NCSD_5403xx : ARRAY  [0 .. 15 ] OF //NC start disable A.no.540300-540315
    BOOL ;
    FdStop_1_5411xx : ARRAY  [0 .. 15 ] OF //Feed stop GEOaxis 1 A.no.541100-541115
    BOOL ;
    FdStop_2_5412xx : ARRAY  [0 .. 15 ] OF //Feed stop GEOaxis 2 A.no.541200-541215
    BOOL ;
    FdStop_3_5413xx : ARRAY  [0 .. 15 ] OF //Feed stop GEOaxis 3 A.no.541300-541315
    BOOL ;
   END_STRUCT ;
   C5 : STRUCT 	//From Channel 5
    FDD_5500xx : ARRAY  [0 .. 15 ] OF //Feed disable A.no.550000-550015
    BOOL ;
    FDD_RID_5501xx : ARRAY  [0 .. 31 ] OF //Feed and read-in disable A.no.550100-550131
    BOOL ;
    RID_5502xx : ARRAY  [0 .. 31 ] OF //Read-in disable A.no.550200-550231
    BOOL ;
    NCSD_5503xx : ARRAY  [0 .. 15 ] OF //NC start disable A.no.550300-550315
    BOOL ;
    FdStop_1_5511xx : ARRAY  [0 .. 15 ] OF //Feed stop GEOaxis 1 A.no.551100-551115
    BOOL ;
    FdStop_2_5512xx : ARRAY  [0 .. 15 ] OF //Feed stop GEOaxis 2 A.no.551200-551215
    BOOL ;
    FdStop_3_5513xx : ARRAY  [0 .. 15 ] OF //Feed stop GEOaxis 3 A.no.551300-551315
    BOOL ;
   END_STRUCT ;
   C6 : STRUCT 	//From Channel 6
    FDD_5600xx : ARRAY  [0 .. 15 ] OF //Feed disable A.no.560000-560015
    BOOL ;
    FDD_RID_5601xx : ARRAY  [0 .. 31 ] OF //Feed and read-in disable A.no.560100-560131
    BOOL ;
    RID_5602xx : ARRAY  [0 .. 31 ] OF //Read-in disable A.no.560200-560231
    BOOL ;
    NCSD_5603xx : ARRAY  [0 .. 15 ] OF //NC start disable A.no.560300-560315
    BOOL ;
    FdStop_1_5611xx : ARRAY  [0 .. 15 ] OF //Feed stop GEOaxis 1 A.no.561100-561115
    BOOL ;
    FdStop_2_5612xx : ARRAY  [0 .. 15 ] OF //Feed stop GEOaxis 2 A.no.561200-561215
    BOOL ;
    FdStop_3_5613xx : ARRAY  [0 .. 15 ] OF //Feed stop GEOaxis 3 A.no.561300-561315
    BOOL ;
   END_STRUCT ;
   C7 : STRUCT 	//From Channel 7
    FDD_5700xx : ARRAY  [0 .. 15 ] OF //Feed disable A.no.570000-570015
    BOOL ;
    FDD_RID_5701xx : ARRAY  [0 .. 31 ] OF //Feed and read-in disable A.no.570100-570131
    BOOL ;
    RID_5702xx : ARRAY  [0 .. 31 ] OF //Read-in disable A.no.570200-570231
    BOOL ;
    NCSD_5703xx : ARRAY  [0 .. 15 ] OF //NC start disable A.no.570300-570315
    BOOL ;
    FdStop_1_5711xx : ARRAY  [0 .. 15 ] OF //Feed stop GEOaxis 1 A.no.571100-511115
    BOOL ;
    FdStop_2_5712xx : ARRAY  [0 .. 15 ] OF //Feed stop GEOaxis 2 A.no.571200-511215
    BOOL ;
    FdStop_3_5713xx : ARRAY  [0 .. 15 ] OF //Feed stop GEOaxis 3 A.no.571300-511315
    BOOL ;
   END_STRUCT ;
   C8 : STRUCT 	//From Channel 8
    FDD_5800xx : ARRAY  [0 .. 15 ] OF //Feed disable A.no.580000-580015
    BOOL ;
    FDD_RID_5801xx : ARRAY  [0 .. 31 ] OF //Feed and read-in disable A.no.580100-510131
    BOOL ;
    RID_5802xx : ARRAY  [0 .. 31 ] OF //Read-in disable A.no.580200-580231
    BOOL ;
    NCSD_5803xx : ARRAY  [0 .. 15 ] OF //NC start disable A.no.580300-580315
    BOOL ;
    FdStop_1_5811xx : ARRAY  [0 .. 15 ] OF //Feed stop GEOaxis 1 A.no.581100-511115
    BOOL ;
    FdStop_2_5812xx : ARRAY  [0 .. 15 ] OF //Feed stop GEOaxis 2 A.no.581200-511215
    BOOL ;
    FdStop_3_5813xx : ARRAY  [0 .. 15 ] OF //Feed stop GEOaxis 3 A.no.581300-511315
    BOOL ;
   END_STRUCT ;
   _1FdStop6001xx : ARRAY  [0 .. 15 ] OF //Feed stop axis/spindle 1
   BOOL ;
   _2FdStop6002xx : ARRAY  [0 .. 15 ] OF //Feed stop axis/spindle 2
   BOOL ;
   _3FdStop6003xx : ARRAY  [0 .. 15 ] OF //Feed stop axis/spindle 3
   BOOL ;
   _4FdStop6004xx : ARRAY  [0 .. 15 ] OF //Feed stop axis/spindle 4
   BOOL ;
   _5FdStop6005xx : ARRAY  [0 .. 15 ] OF //Feed stop axis/spindle 5
   BOOL ;
   _6FdStop6006xx : ARRAY  [0 .. 15 ] OF //Feed stop axis/spindle 6
   BOOL ;
   _7FdStop6007xx : ARRAY  [0 .. 15 ] OF //Feed stop axis/spindle 7
   BOOL ;
   _8FdStop6008xx : ARRAY  [0 .. 15 ] OF //Feed stop axis/spindle 8
   BOOL ;
   _9FdStop6009xx : ARRAY  [0 .. 15 ] OF //Feed stop axis/spindle 9
   BOOL ;
   _10FdStop6010xx : ARRAY  [0 .. 15 ] OF //Feed stop axis/spindle 10
   BOOL ;
   _11FdStop6011xx : ARRAY  [0 .. 15 ] OF //Feed stop axis/spindle 11
   BOOL ;
   _12FdStop6012xx : ARRAY  [0 .. 15 ] OF //Feed stop axis/spindle 12
   BOOL ;
   _13FdStop6013xx : ARRAY  [0 .. 15 ] OF //Feed stop axis/spindle 13
   BOOL ;
   _14FdStop6014xx : ARRAY  [0 .. 15 ] OF //Feed stop axis/spindle 14
   BOOL ;
   _15FdStop6015xx : ARRAY  [0 .. 15 ] OF //Feed stop axis/spindle 15
   BOOL ;
   _16FdStop6016xx : ARRAY  [0 .. 15 ] OF //Feed stop axis/spindle 16
   BOOL ;
   _17FdStop6017xx : ARRAY  [0 .. 15 ] OF //Feed stop axis/spindle 17
   BOOL ;
   _18FdStop6018xx : ARRAY  [0 .. 15 ] OF //Feed stop axis/spindle 18
   BOOL ;
   A7000xx : ARRAY  [0 .. 63 ] OF //Alarm 700000-700063 (user area 0)
   BOOL ;
   A7001xx : ARRAY  [0 .. 63 ] OF //Alarm 700100-700163 (user area 1)
   BOOL ;
   A7002xx : ARRAY  [0 .. 63 ] OF //Alarm 700200-700263 (user area 2)
   BOOL ;
   A7003xx : ARRAY  [0 .. 63 ] OF //Alarm 700300-700363 (user area 3)
   BOOL ;
   A7004xx : ARRAY  [0 .. 63 ] OF //Alarm 700400-700463 (user area 4)
   BOOL ;
   A7005xx : ARRAY  [0 .. 63 ] OF //Alarm 700500-700563 (user area 5
   BOOL ;
   A7006xx : ARRAY  [0 .. 63 ] OF //Alarm 700600-700663 (user area 6)
   BOOL ;
   A7007xx : ARRAY  [0 .. 63 ] OF //Alarm 700700-700763 (user area 7)
   BOOL ;
   A7008xx : ARRAY  [0 .. 63 ] OF //Alarm 700800-700863 (user area 8)
   BOOL ;
   A7009xx : ARRAY  [0 .. 63 ] OF //Alarm 700900-700963 (user area 9)
   BOOL ;
  END_STRUCT ;	
END_TYPE

TYPE UDT 10
VERSION : 0.0
  STRUCT
   A_Disabl_Inp1 : BOOL ;	//Disable digi. NCK input 1
   A_Disabl_Inp2 : BOOL ;	//Disable digi. NCK input 2
   A_Disabl_Inp3 : BOOL ;	//Disable digi. NCK input 3
   A_Disabl_Inp4 : BOOL ;	//Disable digi. NCK input 4
   A_Disabl_Inp5 : BOOL ;	//Disable digi. NCK input 5
   A_Disabl_Inp6 : BOOL ;	//Disable digi. NCK input 6
   A_Disabl_Inp7 : BOOL ;	//Disable digi. NCK input 7
   A_Disabl_Inp8 : BOOL ;	//Disable digi. NCK input 8
   A_Set_Inp1 : BOOL ;	//Set digi. NCK input 1
   A_Set_Inp2 : BOOL ;	//Set digi. NCK input 2
   A_Set_Inp3 : BOOL ;	//Set digi. NCK input 3
   A_Set_Inp4 : BOOL ;	//Set digi. NCK input 4
   A_Set_Inp5 : BOOL ;	//Set digi. NCK input 5
   A_Set_Inp6 : BOOL ;	//Set digi. NCK input 6
   A_Set_Inp7 : BOOL ;	//Set digi. NCK input 7
   A_Set_Inp8 : BOOL ;	//Set digi. NCK input 8
   f0_f15 : ARRAY  [0 .. 15 ] OF BOOL ;	//Reserved
   A_Disabl_Out1 : BOOL ;	//Disable digi. NCK output 1
   A_Disabl_Out2 : BOOL ;	//Disable digi. NCK output 2
   A_Disabl_Out3 : BOOL ;	//Disable digi. NCK output 3
   A_Disabl_Out4 : BOOL ;	//Disable digi. NCK output 4
   A_Disabl_Out5 : BOOL ;	//Disable digi. NCK output 5
   A_Disabl_Out6 : BOOL ;	//Disable digi. NCK output 6
   A_Disabl_Out7 : BOOL ;	//Disable digi. NCK output 7
   A_Disabl_Out8 : BOOL ;	//Disable digi. NCK output 8
   A_OvMask_Out1 : BOOL ;	//Overwrite mask of digi. output 1
   A_OvMask_Out2 : BOOL ;	//Overwrite mask of digi. output 2
   A_OvMask_Out3 : BOOL ;	//Overwrite mask of digi. output 3
   A_OvMask_Out4 : BOOL ;	//Overwrite mask of digi. output 4
   A_OvMask_Out5 : BOOL ;	//Overwrite mask of digi. output 5
   A_OvMask_Out6 : BOOL ;	//Overwrite mask of digi. output 6
   A_OvMask_Out7 : BOOL ;	//Overwrite mask of digi. output 7
   A_OvMask_Out8 : BOOL ;	//Overwrite mask of digi. output 8
   A_Set_Out1 : BOOL ;	//Set digi. NCK output 1
   A_Set_Out2 : BOOL ;	//Set digi. NCK output 2
   A_Set_Out3 : BOOL ;	//Set digi. NCK output 3
   A_Set_Out4 : BOOL ;	//Set digi. NCK output 4
   A_Set_Out5 : BOOL ;	//Set digi. NCK output 5
   A_Set_Out6 : BOOL ;	//Set digi. NCK output 6
   A_Set_Out7 : BOOL ;	//Set digi. NCK output 7
   A_Set_Out8 : BOOL ;	//Set digi. NCK output 8
   A_InMask_Out1 : BOOL ;	//Input mask of digi. output 1
   A_InMask_Out2 : BOOL ;	//Input mask of digi. output 2
   A_InMask_Out3 : BOOL ;	//Input mask of digi. output 3
   A_InMask_Out4 : BOOL ;	//Input mask of digi. output 4
   A_InMask_Out5 : BOOL ;	//Input mask of digi. output 5
   A_InMask_Out6 : BOOL ;	//Input mask of digi. output 6
   A_InMask_Out7 : BOOL ;	//Input mask of digi. output 7
   A_InMask_Out8 : BOOL ;	//Input mask of digi. output 8
   MCP1AxisTbl : ARRAY  [1 .. 22 ] OF BYTE  := B#16#1, B#16#2, B#16#3, B#16#4, B#16#5, B#16#6, B#16#7, B#16#8, B#16#9, B#16#A, B#16#B, B#16#C;	//Axis No. Table MCP1
   MCP1MaxAxis : WORD ;	//max. of Axisno, must be smaller or equal gp_par.MaxAxis
   MCP2AxisTbl : ARRAY  [1 .. 22 ] OF BYTE  := B#16#1, B#16#2, B#16#3, B#16#4, B#16#5, B#16#6, B#16#7, B#16#8, B#16#9, B#16#A, B#16#B, B#16#C;	//Axis No. Table MCP2
   MCP2MaxAxis : WORD ;	//max. of Axisno, must be smaller or equal gp_par.MaxAxis
   f56_0 : BOOL ;
   A_EMERGENCY : BOOL ;	//Emergency stop
   A_EMERGENCY_Ackn : BOOL ;	//Acknowledge emergency stop
   f56_3 : BOOL ;
   A_Keyswitch0 : BOOL ;	//Keyswitch position 0
   A_Keyswitch1 : BOOL ;	//Keyswitch position 1
   A_Keyswitch2 : BOOL ;	//Keyswitch position 2
   A_Keyswitch3 : BOOL ;	//Keyswitch position 3
   A_IncInModeGroup : BOOL ;	//INC inputs in mode group area active
   f57_1 : BOOL ;
   f57_2 : BOOL ;
   A_PCshutdown : BOOL ;	//PC shutdown 840Di
   f57_4 : BOOL ;
   f57_5 : BOOL ;
   f57_6 : BOOL ;
   f57_7 : BOOL ;
   A_CollCheckOff : BOOL ;	//Collisions Check Off
   f58_1 : BOOL ;
   f58_2 : BOOL ;
   f58_3 : BOOL ;
   f58_4 : BOOL ;
   f58_5 : BOOL ;
   f58_6 : BOOL ;
   f58_7 : BOOL ;
   f59 : BYTE ;
   E_ActVal_In1 : BOOL ;	//Actual value of digi. NCK input 1
   E_ActVal_In2 : BOOL ;	//Actual value of digi. NCK input 2
   E_ActVal_In3 : BOOL ;	//Actual value of digi. NCK input 3
   E_ActVal_In4 : BOOL ;	//Actual value of digi. NCK input 4
   f60_4 : BOOL ;
   f60_5 : BOOL ;
   f60_6 : BOOL ;
   f60_7 : BOOL ;
   f61_f62 : ARRAY  [61 .. 61 ] OF BYTE ;
   E_Setpoint_Out1 : BOOL ;	//Setpoint of digi. NCK output 1
   E_Setpoint_Out2 : BOOL ;	//Setpoint of digi. NCK output 2
   E_Setpoint_Out3 : BOOL ;	//Setpoint of digi. NCK output 3
   E_Setpoint_Out4 : BOOL ;	//Setpoint of digi. NCK output 4
   E_Setpoint_Out5 : BOOL ;	//Setpoint of digi. NCK output 5
   E_Setpoint_Out6 : BOOL ;	//Setpoint of digi. NCK output 6
   E_Setpoint_Out7 : BOOL ;	//Setpoint of digi. NCK output 7
   E_Setpoint_Out8 : BOOL ;	//Setpoint of digi. NCK output 8
   f65_f67 : ARRAY  [65 .. 66 ] OF BYTE ;
   E_HW1_moved : BYTE ;	//Handwheel 1 moved
   E_HW2_moved : BYTE ;	//Handwheel 2 moved
   E_HW3_moved : BYTE ;	//Handwheel 3 moved
   E_CounterInchMetr : BYTE ;	//Modification counter inch/metric system of units
   E_MCP1AxisValid : BOOL ;	//from HT6
   E_MCP1WCS : BOOL ;	//from HT6
   f72_2 : BOOL ;
   f72_3 : BOOL ;
   f72_4 : BOOL ;
   f72_5 : BOOL ;
   f72_6 : BOOL ;
   E_MCP1AxKeyDisp : BOOL ;	//Mcp1 Axis Key Displayed
   E_MCP2AxisValid : BOOL ;	//from HT6
   E_MCP2WCS : BOOL ;	//from HT6
   f73_2 : BOOL ;
   f73_3 : BOOL ;
   f73_4 : BOOL ;
   f73_5 : BOOL ;
   f73_6 : BOOL ;
   E_MCP2AxKeyDisp : BOOL ;	//Mcp2 Axis Key Displayed
   MCP1AxisFromHMI : ARRAY  [1 .. 6 ] OF BYTE ;	//Axistable from HT6
   MCP2AxisFromHMI : ARRAY  [1 .. 6 ] OF BYTE ;	//Axistable from HT6
   res86 : WORD ;
   res88 : BYTE ;
   res89 : BYTE ;
   epsToPlc : BYTE ;
   epsFromPlc : BYTE ;
   MpiDpOk : BOOL ;	//Slaves on MPI/DP Ok
   DpOk : BOOL ;	//Slaves on DP Ok
   f92_2 : BOOL ;
   f92_3 : BOOL ;
   f92_4 : BOOL ;
   f92_5 : BOOL ;
   f92_6 : BOOL ;
   f92_7 : BOOL ;
   f93 : BYTE ;
   f94 : BYTE ;
   f95 : BYTE ;
   E_LanguageID : BYTE ;	// LanguageID on HMI
   E_Chan_HW1_A : BOOL ;	//Channel number for handwheel1 A
   E_Chan_HW1_B : BOOL ;	//Channel number for handwheel1 B
   E_Chan_HW1_C : BOOL ;	//Channel number for handwheel1 C
   E_Chan_HW1_D : BOOL ;	//Channel number for handwheel1 D
   f97_4 : BOOL ;
   f97_5 : BOOL ;
   f97_6 : BOOL ;
   f97_7 : BOOL ;
   E_Chan_HW2_A : BOOL ;	//Channel number for handwheel2 A
   E_Chan_HW2_B : BOOL ;	//Channel number for handwheel2 B
   E_Chan_HW2_C : BOOL ;	//Channel number for handwheel2 C
   E_Chan_HW2_D : BOOL ;	//Channel number for handwheel2 D
   f98_4 : BOOL ;
   f98_5 : BOOL ;
   f98_6 : BOOL ;
   f98_7 : BOOL ;
   E_Chan_HW3_A : BOOL ;	//Channel number for handwheel3 A
   E_Chan_HW3_B : BOOL ;	//Channel number for handwheel3 B
   E_Chan_HW3_C : BOOL ;	//Channel number for handwheel3 C
   E_Chan_HW3_D : BOOL ;	//Channel number for handwheel3 D
   f99_4 : BOOL ;
   f99_5 : BOOL ;
   f99_6 : BOOL ;
   f99_7 : BOOL ;
   E_Ax_A_HW1 : BOOL ;	//Axis number for handwheel1 A
   E_Ax_B_HW1 : BOOL ;	//Axis number for handwheel1 B
   E_Ax_C_HW1 : BOOL ;	//Axis number for handwheel1 C
   E_Ax_D_HW1 : BOOL ;	//Axis number for handwheel1 D
   E_Ax_E_HW1 : BOOL ;	//Axis number for handwheel1 E
   E_CHW_sel1 : BOOL ;	//Contour handwheel selected
   E_HW_sel1 : BOOL ;	//Handwheel selected
   E_Mach_Ax1 : BOOL ;	//Machine axis
   E_Ax_A_HW2 : BOOL ;	//Axis number for handwheel2 A
   E_Ax_B_HW2 : BOOL ;	//Axis number for handwheel2 B
   E_Ax_C_HW2 : BOOL ;	//Axis number for handwheel2 C
   E_Ax_D_HW2 : BOOL ;	//Axis number for handwheel2 D
   E_Ax_E_HW2 : BOOL ;	//Axis number for handwheel2 E
   E_CHW_sel2 : BOOL ;	//Contour handwheel selected
   E_HW_sel2 : BOOL ;	//Handwheel selected
   E_Mach_Ax2 : BOOL ;	//Machine axis
   E_Ax_A_HW3 : BOOL ;	//Axis number for handwheel3 A
   E_Ax_B_HW3 : BOOL ;	//Axis number for handwheel3 B
   E_Ax_C_HW3 : BOOL ;	//Axis number for handwheel3 C
   E_Ax_D_HW3 : BOOL ;	//Axis number for handwheel3 D
   E_Ax_E_HW3 : BOOL ;	//Axis number for handwheel3 E
   E_CHW_sel3 : BOOL ;	//Contour handwheel selected
   E_HW_sel3 : BOOL ;	//Handwheel selected
   E_Mach_Ax3 : BOOL ;	//Machine axis
   E_RemDiag : BOOL ;	//Remote Diagnostic
   f103_1 : BOOL ;
   f103_2 : BOOL ;
   f103_3 : BOOL ;
   f103_4 : BOOL ;
   E_ATready : BOOL ;	//AT-box ready
   E_MMCTemp : BOOL ;	//MMC temperature limit
   E_MMCBatt : BOOL ;	//MMC 101/102 battery alarm
   E_MCP1ready : BOOL ;	//MCP1 ready;
   E_MCP2ready : BOOL ;	//MCP2 ready;
   E_BHGready : BOOL ;	//BHG ready;
   f104_3 : BOOL ;
   f104_4 : BOOL ;
   f104_5 : BOOL ;
   E_FirstOB1 : BOOL ;	//This bit is on for the first OB1 cycle
   E_NCKready : BOOL ;	//NCK CPU ready
   E_CancelToolCmd : BOOL ;	//Terminate canceled tool command
   f105_1 : BOOL ;
   f105_2 : BOOL ;
   f105_3 : BOOL ;
   f105_4 : BOOL ;
   f105_5 : BOOL ;
   f105_6 : BOOL ;
   f105_7 : BOOL ;
   E_CollCheckOff : BOOL ;	//CollisionsCheck Off
   E_EMSTOP : BOOL ;	//EMERGENCY STOP active
   f106_2 : BOOL ;
   f106_3 : BOOL ;
   f106_4 : BOOL ;
   f106_5 : BOOL ;
   f106_6 : BOOL ;
   f106_7 : BOOL ;
   E_InspProbe1 : BOOL ;	//Inspection probe 1 actuated
   E_InspProbe2 : BOOL ;	//Inspection probe 2 actuated
   f107_2 : BOOL ;
   f107_3 : BOOL ;
   f107_4 : BOOL ;
   f107_5 : BOOL ;
   E_NCU_LinkActive : BOOL ;	//NCU link active
   E_SystemInchDim : BOOL ;	//System inch dimension
   f108_0 : BOOL ;
   E_MMC2Ready : BOOL ;	//MMC2-CPU ready
   E_MMCMPIready : BOOL ;	//MMC1-CPU on MPI ready
   E_MMCBTSSready : BOOL ;	//MMC1-CPU on BTSS ready
   f108_4 : BOOL ;
   E_DrivesInCylOp : BOOL ;	//Drives in cylindric operation
   E_611Dready : BOOL ;	//611D ready
   E_NCready : BOOL ;
   E_NCKalarm : BOOL ;	//NCK alarm present
   f109_1 : BOOL ;
   f109_2 : BOOL ;
   f109_3 : BOOL ;
   A_PC_OSfault : BOOL ;	//PC operating system fault, 840Di
   E_HTempAlarm : BOOL ;	//Heat sink temperature alarm NCU 573
   E_ATempAlarm : BOOL ;	//Air temperature alarm
   E_BattAlarm : BOOL ;	//NCK battery alarm
   E_SWCamMinus : ARRAY  [0 .. 31 ] OF BOOL ;	//Software cams minus [0..31]
   E_SWCamPlus : ARRAY  [0 .. 31 ] OF BOOL ;	//Software cams plus [0..31]
   f118_f121 : ARRAY  [0 .. 3 ] OF BYTE ;
   A_Disabl_Inp9 : BOOL ;	//Disable digi. NCK input 9
   A_Disabl_Inp10 : BOOL ;	//Disable digi. NCK input 10
   A_Disabl_Inp11 : BOOL ;	//Disable digi. NCK input 11
   A_Disabl_Inp12 : BOOL ;	//Disable digi. NCK input 12
   A_Disabl_Inp13 : BOOL ;	//Disable digi. NCK input 13
   A_Disabl_Inp14 : BOOL ;	//Disable digi. NCK input 14
   A_Disabl_Inp15 : BOOL ;	//Disable digi. NCK input 15
   A_Disabl_Inp16 : BOOL ;	//Disable digi. NCK input 16
   A_Set_Inp9 : BOOL ;	//Set digi. NCK input 9
   A_Set_Inp10 : BOOL ;	//Set digi. NCK input 10
   A_Set_Inp11 : BOOL ;	//Set digi. NCK input 11
   A_Set_Inp12 : BOOL ;	//Set digi. NCK input 12
   A_Set_Inp13 : BOOL ;	//Set digi. NCK input 13
   A_Set_Inp14 : BOOL ;	//Set digi. NCK input 14
   A_Set_Inp15 : BOOL ;	//Set digi. NCK input 15
   A_Set_Inp16 : BOOL ;	//Set digi. NCK input 16
   A_Disabl_Inp17 : BOOL ;	//Disable digi. NCK input 17
   A_Disabl_Inp18 : BOOL ;	//Disable digi. NCK input 18
   A_Disabl_Inp19 : BOOL ;	//Disable digi. NCK input 19
   A_Disabl_Inp20 : BOOL ;	//Disable digi. NCK input 20
   A_Disabl_Inp21 : BOOL ;	//Disable digi. NCK input 21
   A_Disabl_Inp22 : BOOL ;	//Disable digi. NCK input 22
   A_Disabl_Inp23 : BOOL ;	//Disable digi. NCK input 23
   A_Disabl_Inp24 : BOOL ;	//Disable digi. NCK input 24
   A_Set_Inp17 : BOOL ;	//Set digi. NCK input 17
   A_Set_Inp18 : BOOL ;	//Set digi. NCK input 18
   A_Set_Inp19 : BOOL ;	//Set digi. NCK input 19
   A_Set_Inp20 : BOOL ;	//Set digi. NCK input 20
   A_Set_Inp21 : BOOL ;	//Set digi. NCK input 21
   A_Set_Inp22 : BOOL ;	//Set digi. NCK input 22
   A_Set_Inp23 : BOOL ;	//Set digi. NCK input 23
   A_Set_Inp24 : BOOL ;	//Set digi. NCK input 24
   A_Disabl_Inp25 : BOOL ;	//Disable digi. NCK input 25
   A_Disabl_Inp26 : BOOL ;	//Disable digi. NCK input 26
   A_Disabl_Inp27 : BOOL ;	//Disable digi. NCK input 27
   A_Disabl_Inp28 : BOOL ;	//Disable digi. NCK input 28
   A_Disabl_Inp29 : BOOL ;	//Disable digi. NCK input 29
   A_Disabl_Inp30 : BOOL ;	//Disable digi. NCK input 30
   A_Disabl_Inp31 : BOOL ;	//Disable digi. NCK input 31
   A_Disabl_Inp32 : BOOL ;	//Disable digi. NCK input 32
   A_Set_Inp25 : BOOL ;	//Set digi. NCK input 25
   A_Set_Inp26 : BOOL ;	//Set digi. NCK input 26
   A_Set_Inp27 : BOOL ;	//Set digi. NCK input 27
   A_Set_Inp28 : BOOL ;	//Set digi. NCK input 28
   A_Set_Inp29 : BOOL ;	//Set digi. NCK input 29
   A_Set_Inp30 : BOOL ;	//Set digi. NCK input 30
   A_Set_Inp31 : BOOL ;	//Set digi. NCK input 31
   A_Set_Inp32 : BOOL ;	//Set digi. NCK input 32
   A_Disabl_Inp33 : BOOL ;	//Disable digi. NCK input 33
   A_Disabl_Inp34 : BOOL ;	//Disable digi. NCK input 34
   A_Disabl_Inp35 : BOOL ;	//Disable digi. NCK input 35
   A_Disabl_Inp36 : BOOL ;	//Disable digi. NCK input 36
   A_Disabl_Inp37 : BOOL ;	//Disable digi. NCK input 37
   A_Disabl_Inp38 : BOOL ;	//Disable digi. NCK input 38
   A_Disabl_Inp39 : BOOL ;	//Disable digi. NCK input 39
   A_Disabl_Inp40 : BOOL ;	//Disable digi. NCK input 40
   A_Set_Inp33 : BOOL ;	//Set digi. NCK input 33
   A_Set_Inp34 : BOOL ;	//Set digi. NCK input 34
   A_Set_Inp35 : BOOL ;	//Set digi. NCK input 35
   A_Set_Inp36 : BOOL ;	//Set digi. NCK input 36
   A_Set_Inp37 : BOOL ;	//Set digi. NCK input 37
   A_Set_Inp38 : BOOL ;	//Set digi. NCK input 38
   A_Set_Inp39 : BOOL ;	//Set digi. NCK input 39
   A_Set_Inp40 : BOOL ;	//Set digi. NCK input 40
   A_Disabl_Out9 : BOOL ;	//Disable digi. NCK output 9
   A_Disabl_Out10 : BOOL ;	//Disable digi. NCK output 10
   A_Disabl_Out11 : BOOL ;	//Disable digi. NCK output 11
   A_Disabl_Out12 : BOOL ;	//Disable digi. NCK output 12
   A_Disabl_Out13 : BOOL ;	//Disable digi. NCK output 13
   A_Disabl_Out14 : BOOL ;	//Disable digi. NCK output 14
   A_Disabl_Out15 : BOOL ;	//Disable digi. NCK output 15
   A_Disabl_Out16 : BOOL ;	//Disable digi. NCK output 16
   A_OvMask_Out9 : BOOL ;	//Overwrite mask of digi. output 9
   A_OvMask_Out10 : BOOL ;	//Overwrite mask of digi. output 10
   A_OvMask_Out11 : BOOL ;	//Overwrite mask of digi. output 11
   A_OvMask_Out12 : BOOL ;	//Overwrite mask of digi. output 12
   A_OvMask_Out13 : BOOL ;	//Overwrite mask of digi. output 13
   A_OvMask_Out14 : BOOL ;	//Overwrite mask of digi. output 14
   A_OvMask_Out15 : BOOL ;	//Overwrite mask of digi. output 15
   A_OvMask_Out16 : BOOL ;	//Overwrite mask of digi. output 16
   A_Setval_Out9 : BOOL ;	//Set value digi. NCK output 9
   A_Setval_Out10 : BOOL ;	//Set value digi. NCK output 10
   A_Setval_Out11 : BOOL ;	//Set value digi. NCK output 11
   A_Setval_Out12 : BOOL ;	//Set value digi. NCK output 12
   A_Setval_Out13 : BOOL ;	//Set value digi. NCK output 13
   A_Setval_Out14 : BOOL ;	//Set value digi. NCK output 14
   A_Setval_Out15 : BOOL ;	//Set value digi. NCK output 15
   A_Setval_Out16 : BOOL ;	//Set value digi. NCK output 16
   A_InMask_Out9 : BOOL ;	//Input mask of digi. output 9
   A_InMask_Out10 : BOOL ;	//Input mask of digi. output 10
   A_InMask_Out11 : BOOL ;	//Input mask of digi. output 11
   A_InMask_Out12 : BOOL ;	//Input mask of digi. output 12
   A_InMask_Out13 : BOOL ;	//Input mask of digi. output 13
   A_InMask_Out14 : BOOL ;	//Input mask of digi. output 14
   A_InMask_Out15 : BOOL ;	//Input mask of digi. output 15
   A_InMask_Out16 : BOOL ;	//Input mask of digi. output 16
   A_Disabl_Out17 : BOOL ;	//Disable digi. NCK output 17
   A_Disabl_Out18 : BOOL ;	//Disable digi. NCK output 18
   A_Disabl_Out19 : BOOL ;	//Disable digi. NCK output 19
   A_Disabl_Out20 : BOOL ;	//Disable digi. NCK output 20
   A_Disabl_Out21 : BOOL ;	//Disable digi. NCK output 21
   A_Disabl_Out22 : BOOL ;	//Disable digi. NCK output 22
   A_Disabl_Out23 : BOOL ;	//Disable digi. NCK output 23
   A_Disabl_Out24 : BOOL ;	//Disable digi. NCK output 24
   A_OvMask_Out17 : BOOL ;	//Overwrite mask of digi. output 17
   A_OvMask_Out18 : BOOL ;	//Overwrite mask of digi. output 18
   A_OvMask_Out19 : BOOL ;	//Overwrite mask of digi. output 19
   A_OvMask_Out20 : BOOL ;	//Overwrite mask of digi. output 20
   A_OvMask_Out21 : BOOL ;	//Overwrite mask of digi. output 21
   A_OvMask_Out22 : BOOL ;	//Overwrite mask of digi. output 22
   A_OvMask_Out23 : BOOL ;	//Overwrite mask of digi. output 23
   A_OvMask_Out24 : BOOL ;	//Overwrite mask of digi. output 24
   A_Setval_Out17 : BOOL ;	//Set value digi. NCK output 17
   A_Setval_Out18 : BOOL ;	//Set value digi. NCK output 18
   A_Setval_Out19 : BOOL ;	//Set value digi. NCK output 19
   A_Setval_Out20 : BOOL ;	//Set value digi. NCK output 20
   A_Setval_Out21 : BOOL ;	//Set value digi. NCK output 21
   A_Setval_Out22 : BOOL ;	//Set value digi. NCK output 22
   A_Setval_Out23 : BOOL ;	//Set value digi. NCK output 23
   A_Setval_Out24 : BOOL ;	//Set value digi. NCK output 24
   A_InMask_Out17 : BOOL ;	//Input mask of digi. output 17
   A_InMask_Out18 : BOOL ;	//Input mask of digi. output 18
   A_InMask_Out19 : BOOL ;	//Input mask of digi. output 19
   A_InMask_Out20 : BOOL ;	//Input mask of digi. output 20
   A_InMask_Out21 : BOOL ;	//Input mask of digi. output 21
   A_InMask_Out22 : BOOL ;	//Input mask of digi. output 22
   A_InMask_Out23 : BOOL ;	//Input mask of digi. output 23
   A_InMask_Out24 : BOOL ;	//Input mask of digi. output 24
   A_Disabl_Out25 : BOOL ;	//Disable digi. NCK output 25
   A_Disabl_Out26 : BOOL ;	//Disable digi. NCK output 26
   A_Disabl_Out27 : BOOL ;	//Disable digi. NCK output 27
   A_Disabl_Out28 : BOOL ;	//Disable digi. NCK output 28
   A_Disabl_Out29 : BOOL ;	//Disable digi. NCK output 29
   A_Disabl_Out30 : BOOL ;	//Disable digi. NCK output 30
   A_Disabl_Out31 : BOOL ;	//Disable digi. NCK output 31
   A_Disabl_Out32 : BOOL ;	//Disable digi. NCK output 32
   A_OvMask_Out25 : BOOL ;	//Overwrite mask of digi. output 25
   A_OvMask_Out26 : BOOL ;	//Overwrite mask of digi. output 26
   A_OvMask_Out27 : BOOL ;	//Overwrite mask of digi. output 27
   A_OvMask_Out28 : BOOL ;	//Overwrite mask of digi. output 28
   A_OvMask_Out29 : BOOL ;	//Overwrite mask of digi. output 29
   A_OvMask_Out30 : BOOL ;	//Overwrite mask of digi. output 30
   A_OvMask_Out31 : BOOL ;	//Overwrite mask of digi. output 31
   A_OvMask_Out32 : BOOL ;	//Overwrite mask of digi. output 32
   A_Setval_Out25 : BOOL ;	//Set value digi. NCK output 25
   A_Setval_Out26 : BOOL ;	//Set value digi. NCK output 26
   A_Setval_Out27 : BOOL ;	//Set value digi. NCK output 27
   A_Setval_Out28 : BOOL ;	//Set value digi. NCK output 28
   A_Setval_Out29 : BOOL ;	//Set value digi. NCK output 29
   A_Setval_Out30 : BOOL ;	//Set value digi. NCK output 30
   A_Setval_Out31 : BOOL ;	//Set value digi. NCK output 31
   A_Setval_Out32 : BOOL ;	//Set value digi. NCK output 32
   A_InMask_Out25 : BOOL ;	//Input mask of digi. output 25
   A_InMask_Out26 : BOOL ;	//Input mask of digi. output 26
   A_InMask_Out27 : BOOL ;	//Input mask of digi. output 27
   A_InMask_Out28 : BOOL ;	//Input mask of digi. output 28
   A_InMask_Out29 : BOOL ;	//Input mask of digi. output 29
   A_InMask_Out30 : BOOL ;	//Input mask of digi. output 30
   A_InMask_Out31 : BOOL ;	//Input mask of digi. output 31
   A_InMask_Out32 : BOOL ;	//Input mask of digi. output 32
   A_Disabl_Out33 : BOOL ;	//Disable digi. NCK output 33
   A_Disabl_Out34 : BOOL ;	//Disable digi. NCK output 34
   A_Disabl_Out35 : BOOL ;	//Disable digi. NCK output 35
   A_Disabl_Out36 : BOOL ;	//Disable digi. NCK output 36
   A_Disabl_Out37 : BOOL ;	//Disable digi. NCK output 37
   A_Disabl_Out38 : BOOL ;	//Disable digi. NCK output 38
   A_Disabl_Out39 : BOOL ;	//Disable digi. NCK output 39
   A_Disabl_Out40 : BOOL ;	//Disable digi. NCK output 40
   A_OvMask_Out33 : BOOL ;	//Overwrite mask of digi. output 33
   A_OvMask_Out34 : BOOL ;	//Overwrite mask of digi. output 34
   A_OvMask_Out35 : BOOL ;	//Overwrite mask of digi. output 35
   A_OvMask_Out36 : BOOL ;	//Overwrite mask of digi. output 36
   A_OvMask_Out37 : BOOL ;	//Overwrite mask of digi. output 37
   A_OvMask_Out38 : BOOL ;	//Overwrite mask of digi. output 38
   A_OvMask_Out39 : BOOL ;	//Overwrite mask of digi. output 39
   A_OvMask_Out40 : BOOL ;	//Overwrite mask of digi. output 40
   A_Setval_out33 : BOOL ;	//Set value digi. NCK output 33
   A_Setval_out34 : BOOL ;	//Set value digi. NCK output 34
   A_Setval_out35 : BOOL ;	//Set value digi. NCK output 35
   A_Setval_out36 : BOOL ;	//Set value digi. NCK output 36
   A_Setval_out37 : BOOL ;	//Set value digi. NCK output 37
   A_Setval_out38 : BOOL ;	//Set value digi. NCK output 38
   A_Setval_out39 : BOOL ;	//Set value digi. NCK output 39
   A_Setval_out40 : BOOL ;	//Set value digi. NCK output 40
   A_InMask_Out33 : BOOL ;	//Input mask of digi. output 33
   A_InMask_Out34 : BOOL ;	//Input mask of digi. output 34
   A_InMask_Out35 : BOOL ;	//Input mask of digi. output 35
   A_InMask_Out36 : BOOL ;	//Input mask of digi. output 36
   A_InMask_Out37 : BOOL ;	//Input mask of digi. output 37
   A_InMask_Out38 : BOOL ;	//Input mask of digi. output 38
   A_InMask_Out39 : BOOL ;	//Input mask of digi. output 39
   A_InMask_Out40 : BOOL ;	//Input mask of digi. output 40
   A_Disabl_anaIn1 : BOOL ;	//Disable analog NCK input 1
   A_Disabl_anaIn2 : BOOL ;	//Disable analog NCK input 2
   A_Disabl_anaIn3 : BOOL ;	//Disable analog NCK input 3
   A_Disabl_anaIn4 : BOOL ;	//Disable analog NCK input 4
   A_Disabl_anaIn5 : BOOL ;	//Disable analog NCK input 5
   A_Disabl_anaIn6 : BOOL ;	//Disable analog NCK input 6
   A_Disabl_anaIn7 : BOOL ;	//Disable analog NCK input 7
   A_Disabl_anaIn8 : BOOL ;	//Disable analog NCK input 8
   A_InMask_anaIn1 : BOOL ;	//Input mask of analog NCK input 1
   A_InMask_anaIn2 : BOOL ;	//Input mask of analog NCK input 2
   A_InMask_anaIn3 : BOOL ;	//Input mask of analog NCK input 3
   A_InMask_anaIn4 : BOOL ;	//Input mask of analog NCK input 4
   A_InMask_anaIn5 : BOOL ;	//Input mask of analog NCK input 5
   A_InMask_anaIn6 : BOOL ;	//Input mask of analog NCK input 6
   A_InMask_anaIn7 : BOOL ;	//Input mask of analog NCK input 7
   A_InMask_anaIn8 : BOOL ;	//Input mask of analog NCK input 8
   A_Setval_anaIn1 : WORD ;	//Set value of analog NCK input 1
   A_Setval_anaIn2 : WORD ;	//Set value of analog NCK input 2
   A_Setval_anaIn3 : WORD ;	//Set value of analog NCK input 3
   A_Setval_anaIn4 : WORD ;	//Set value of analog NCK input 4
   A_Setval_anaIn5 : WORD ;	//Set value of analog NCK input 5
   A_Setval_anaIn6 : WORD ;	//Set value of analog NCK input 6
   A_Setval_anaIn7 : WORD ;	//Set value of analog NCK input 7
   A_Setval_anaIn8 : WORD ;	//Set value of analog NCK input 8
   f164_f165 : INT ;
   A_OvMask_anaOut1 : BOOL ;	//Overwrite mask of analog output 1
   A_OvMask_anaOut2 : BOOL ;	//Overwrite mask of analog output 2
   A_OvMask_anaOut3 : BOOL ;	//Overwrite mask of analog output 3
   A_OvMask_anaOut4 : BOOL ;	//Overwrite mask of analog output 4
   A_OvMask_anaOut5 : BOOL ;	//Overwrite mask of analog output 5
   A_OvMask_anaOut6 : BOOL ;	//Overwrite mask of analog output 6
   A_OvMask_anaOut7 : BOOL ;	//Overwrite mask of analog output 7
   A_OvMask_anaOut8 : BOOL ;	//Overwrite mask of analog output 8
   A_InMask_anaOut1 : BOOL ;	//Input mask of analog NCK output 1
   A_InMask_anaOut2 : BOOL ;	//Input mask of analog NCK output 2
   A_InMask_anaOut3 : BOOL ;	//Input mask of analog NCK output 3
   A_InMask_anaOut4 : BOOL ;	//Input mask of analog NCK output 4
   A_InMask_anaOut5 : BOOL ;	//Input mask of analog NCK output 5
   A_InMask_anaOut6 : BOOL ;	//Input mask of analog NCK output 6
   A_InMask_anaOut7 : BOOL ;	//Input mask of analog NCK output 7
   A_InMask_anaOut8 : BOOL ;	//Input mask of analog NCK output 8
   A_Disabl_anaOut1 : BOOL ;	//Disable analog NCK output 1
   A_Disabl_anaOut2 : BOOL ;	//Disable analog NCK output 2
   A_Disabl_anaOut3 : BOOL ;	//Disable analog NCK output 3
   A_Disabl_anaOut4 : BOOL ;	//Disable analog NCK output 4
   A_Disabl_anaOut5 : BOOL ;	//Disable analog NCK output 5
   A_Disabl_anaOut6 : BOOL ;	//Disable analog NCK output 6
   A_Disabl_anaOut7 : BOOL ;	//Disable analog NCK output 7
   A_Disabl_anaOut8 : BOOL ;	//Disable analog NCK output 8
   f169 : BYTE ;
   A_Setval_anaOut1 : WORD ;	//Set value of analog NCK output 1
   A_Setval_anaOut2 : WORD ;	//Set value of analog NCK output 2
   A_Setval_anaOut3 : WORD ;	//Set value of analog NCK output 3
   A_Setval_anaOut4 : WORD ;	//Set value of analog NCK output 4
   A_Setval_anaOut5 : WORD ;	//Set value of analog NCK output 5
   A_Setval_anaOut6 : WORD ;	//Set value of analog NCK output 6
   A_Setval_anaOut7 : WORD ;	//Set value of analog NCK output 7
   A_Setval_anaOut8 : WORD ;	//Set value of analog NCK output 8
   E_ActVal_In9 : BOOL ;	//Actual value of digi. NCK input 9
   E_ActVal_In10 : BOOL ;	//Actual value of digi. NCK input 10
   E_ActVal_In11 : BOOL ;	//Actual value of digi. NCK input 11
   E_ActVal_In12 : BOOL ;	//Actual value of digi. NCK input 12
   E_ActVal_In13 : BOOL ;	//Actual value of digi. NCK input 13
   E_ActVal_In14 : BOOL ;	//Actual value of digi. NCK input 14
   E_ActVal_In15 : BOOL ;	//Actual value of digi. NCK input 15
   E_ActVal_In16 : BOOL ;	//Actual value of digi. NCK input 16
   E_ActVal_In17 : BOOL ;	//Actual value of digi. NCK input 17
   E_ActVal_In18 : BOOL ;	//Actual value of digi. NCK input 18
   E_ActVal_In19 : BOOL ;	//Actual value of digi. NCK input 19
   E_ActVal_In20 : BOOL ;	//Actual value of digi. NCK input 20
   E_ActVal_In21 : BOOL ;	//Actual value of digi. NCK input 21
   E_ActVal_In22 : BOOL ;	//Actual value of digi. NCK input 22
   E_ActVal_In23 : BOOL ;	//Actual value of digi. NCK input 23
   E_ActVal_In24 : BOOL ;	//Actual value of digi. NCK input 24
   E_ActVal_In25 : BOOL ;	//Actual value of digi. NCK input 25
   E_ActVal_In26 : BOOL ;	//Actual value of digi. NCK input 26
   E_ActVal_In27 : BOOL ;	//Actual value of digi. NCK input 27
   E_ActVal_In28 : BOOL ;	//Actual value of digi. NCK input 28
   E_ActVal_In29 : BOOL ;	//Actual value of digi. NCK input 29
   E_ActVal_In30 : BOOL ;	//Actual value of digi. NCK input 30
   E_ActVal_In31 : BOOL ;	//Actual value of digi. NCK input 31
   E_ActVal_In32 : BOOL ;	//Actual value of digi. NCK input 32
   E_ActVal_In33 : BOOL ;	//Actual value of digi. NCK input 33
   E_ActVal_In34 : BOOL ;	//Actual value of digi. NCK input 34
   E_ActVal_In35 : BOOL ;	//Actual value of digi. NCK input 35
   E_ActVal_In36 : BOOL ;	//Actual value of digi. NCK input 36
   E_ActVal_In37 : BOOL ;	//Actual value of digi. NCK input 37
   E_ActVal_In38 : BOOL ;	//Actual value of digi. NCK input 38
   E_ActVal_In39 : BOOL ;	//Actual value of digi. NCK input 39
   E_ActVal_In40 : BOOL ;	//Actual value of digi. NCK input 40
   E_Setpoint_Out9 : BOOL ;	//Setpoint of digi. NCK output 9
   E_Setpoint_Out10 : BOOL ;	//Setpoint of digi. NCK output 10
   E_Setpoint_Out11 : BOOL ;	//Setpoint of digi. NCK output 11
   E_Setpoint_Out12 : BOOL ;	//Setpoint of digi. NCK output 12
   E_Setpoint_Out13 : BOOL ;	//Setpoint of digi. NCK output 13
   E_Setpoint_Out14 : BOOL ;	//Setpoint of digi. NCK output 14
   E_Setpoint_Out15 : BOOL ;	//Setpoint of digi. NCK output 15
   E_Setpoint_Out16 : BOOL ;	//Setpoint of digi. NCK output 16
   E_Setpoint_Out17 : BOOL ;	//Setpoint of digi. NCK output 17
   E_Setpoint_Out18 : BOOL ;	//Setpoint of digi. NCK output 18
   E_Setpoint_Out19 : BOOL ;	//Setpoint of digi. NCK output 19
   E_Setpoint_Out20 : BOOL ;	//Setpoint of digi. NCK output 20
   E_Setpoint_Out21 : BOOL ;	//Setpoint of digi. NCK output 21
   E_Setpoint_Out22 : BOOL ;	//Setpoint of digi. NCK output 22
   E_Setpoint_Out23 : BOOL ;	//Setpoint of digi. NCK output 23
   E_Setpoint_Out24 : BOOL ;	//Setpoint of digi. NCK output 24
   E_Setpoint_Out25 : BOOL ;	//Setpoint of digi. NCK output 25
   E_Setpoint_Out26 : BOOL ;	//Setpoint of digi. NCK output 26
   E_Setpoint_Out27 : BOOL ;	//Setpoint of digi. NCK output 27
   E_Setpoint_Out28 : BOOL ;	//Setpoint of digi. NCK output 28
   E_Setpoint_Out29 : BOOL ;	//Setpoint of digi. NCK output 29
   E_Setpoint_Out30 : BOOL ;	//Setpoint of digi. NCK output 30
   E_Setpoint_Out31 : BOOL ;	//Setpoint of digi. NCK output 31
   E_Setpoint_Out32 : BOOL ;	//Setpoint of digi. NCK output 32
   E_Setpoint_Out33 : BOOL ;	//Setpoint of digi. NCK output 33
   E_Setpoint_Out34 : BOOL ;	//Setpoint of digi. NCK output 34
   E_Setpoint_Out35 : BOOL ;	//Setpoint of digi. NCK output 35
   E_Setpoint_Out36 : BOOL ;	//Setpoint of digi. NCK output 36
   E_Setpoint_Out37 : BOOL ;	//Setpoint of digi. NCK output 37
   E_Setpoint_Out38 : BOOL ;	//Setpoint of digi. NCK output 38
   E_Setpoint_Out39 : BOOL ;	//Setpoint of digi. NCK output 39
   E_Setpoint_Out40 : BOOL ;	//Setpoint of digi. NCK output 40
   E_ActVal_anaIn1 : WORD ;	//Actual value of analog NCK input 1
   E_ActVal_anaIn2 : WORD ;	//Actual value of analog NCK input 2
   E_ActVal_anaIn3 : WORD ;	//Actual value of analog NCK input 3
   E_ActVal_anaIn4 : WORD ;	//Actual value of analog NCK input 4
   E_ActVal_anaIn5 : WORD ;	//Actual value of analog NCK input 5
   E_ActVal_anaIn6 : WORD ;	//Actual value of analog NCK input 6
   E_ActVal_anaIn7 : WORD ;	//Actual value of analog NCK input 7
   E_ActVal_anaIn8 : WORD ;	//Actual value of analog NCK input 8
   E_SetVal_anaOut1 : WORD ;	//Set value of analog NCK output 1
   E_SetVal_anaOut2 : WORD ;	//Set value of analog NCK output 2
   E_SetVal_anaOut3 : WORD ;	//Set value of analog NCK output 3
   E_SetVal_anaOut4 : WORD ;	//Set value of analog NCK output 4
   E_SetVal_anaOut5 : WORD ;	//Set value of analog NCK output 5
   E_SetVal_anaOut6 : WORD ;	//Set value of analog NCK output 6
   E_SetVal_anaOut7 : WORD ;	//Set value of analog NCK output 7
   E_SetVal_anaOut8 : WORD ;	//Set value of analog NCK output 8
   E_CollCheck : ARRAY  [0 .. 7 ] OF BYTE ;	//CollisionsCheck
   A_CollCheck : ARRAY  [0 .. 7 ] OF BYTE ;	//CollisionsCheck
   E_HW4_moved : BYTE ;	//Handwheel 4 moved
   E_HW5_moved : BYTE ;	//Handwheel 5 moved
   E_HW6_moved : BYTE ;	//Handwheel 6 moved
   E_EHW1_stands : BOOL ;	//Ethernet handwheel 1 stands
   E_EHW2_stands : BOOL ;	//Ethernet handwheel 2 stands
   E_EHW3_stands : BOOL ;	//Ethernet handwheel 3 stands
   E_EHW4_stands : BOOL ;	//Ethernet handwheel 4 stands
   E_EHW5_stands : BOOL ;	//Ethernet handwheel 5 stands
   E_EHW6_stands : BOOL ;	//Ethernet handwheel 6 stands
   f245_6 : BOOL ;
   f245_7 : BOOL ;
   f246 : WORD ;
  END_STRUCT ;	
END_TYPE

TYPE UDT 11
VERSION : 0.0
  STRUCT
   A_AUTO : BOOL ;	//AUTOMATIC mode
   A_MDA : BOOL ;	//MDA mode
   A_JOG : BOOL ;	//JOG mode
   f0_3 : BOOL ;
   A_MCDisable : BOOL ;	//Mode change disable
   A_MGStop : BOOL ;	//Mode group stop
   A_MGStopASp : BOOL ;	//Mode group stop axes plus spindle
   A_MGReset : BOOL ;	//Mode group reset
   A_TEACHIN : BOOL ;	//Machine function TEACH IN
   A_REPOS : BOOL ;	//Machine function REPOS
   A_REF : BOOL ;	//Machine function REF
   f1_3 : BOOL ;
   f1_4 : BOOL ;
   f1_5 : BOOL ;
   A_SingleBlock_B : BOOL ;	// Single block type B
   A_SingleBlock_A : BOOL ;	// Single block type A
   A_INC1 : BOOL ;	//INC1
   A_INC10 : BOOL ;	//INC10
   A_INC100 : BOOL ;	//INC100
   A_INC1000 : BOOL ;	//INC1000
   A_INC10000 : BOOL ;	//INC10000
   A_INCVar : BOOL ;	//INC variable
   f3 : BYTE ;
   E_MMC_AUTO : BOOL ;	//MMC Strobe AUTOMATIC mode
   E_MMC_MDA : BOOL ;	//MMC Strobe MDA mode
   E_MMC_JOG : BOOL ;	//MMC Strobe JOG mode
   f4_3 : BOOL ;
   f4_4 : BOOL ;
   f4_5 : BOOL ;
   f4_6 : BOOL ;
   f4_7 : BOOL ;
   E_MMC_TEACHIN : BOOL ;	//MMC Strobe machine function TEACH IN
   E_MMC_REPOS : BOOL ;	//MMC Strobe machine function REPOS
   E_MMC_REF : BOOL ;	//MMC Strobe Machine function REF
   f5_3 : BOOL ;
   f5_4 : BOOL ;
   f5_5 : BOOL ;
   f5_6 : BOOL ;
   f5_7 : BOOL ;
   E_AUTO : BOOL ;	//Active AUTOMATIC mode
   E_MDA : BOOL ;	//Active MDA mode
   E_JOG : BOOL ;	//Active JOG mode
   E_MGOK : BOOL ;	//Mode group ready
   E_MGreseted : BOOL ;	// Mode Group reseted
   E_NCKintJOG : BOOL ;	// NCK internal JOG active
   f6_6 : BOOL ;
   E_ChanReset : BOOL ;	//All channels in reset state
   E_TEACHIN : BOOL ;	//Active machine function TEACH IN
   E_REPOS : BOOL ;	//Active machine function REPOS
   E_REF : BOOL ;	//Active Machine function REF
   f7_3 : BOOL ;
   f7_4 : BOOL ;
   f7_5 : BOOL ;
   f7_6 : BOOL ;
   f7_7 : BOOL ;
   E_INC1 : BOOL ;	//INC1
   E_INC10 : BOOL ;	//INC10
   E_INC100 : BOOL ;	//INC100
   E_INC1000 : BOOL ;	//INC1000
   E_INC10000 : BOOL ;	//INC10000
   E_INCVar : BOOL ;	//INC variable
   f8_6 : BOOL ;
   f8_7 : BOOL ;
   f9 : BYTE ;
   f10 : ARRAY  [10 .. 19 ] OF BYTE ;
   MG : ARRAY  [2 .. 10 ] OF STRUCT
    A_AUTO : BOOL ;	//AUTOMATIC mode
    A_MDA : BOOL ;	//MDA mode
    A_JOG : BOOL ;	//JOG mode
    f0_3 : BOOL ;
    A_MCDisable : BOOL ;	//Mode change disable
    A_MGStop : BOOL ;	//Mode group stop
    A_MGStopASp : BOOL ;	//Mode group stop axes plus spindle
    A_MGReset : BOOL ;	//Mode group reset
    A_TEACHIN : BOOL ;	//Machine function TEACH IN
    A_REPOS : BOOL ;	//Machine function REPOS
    A_REF : BOOL ;	//Machine function REF
    f1_3 : BOOL ;
    f1_4 : BOOL ;
    f1_5 : BOOL ;
    A_SingleBlock_B : BOOL ;	// Single block type B
    A_SingleBlock_A : BOOL ;	// Single block type A
    A_INC1 : BOOL ;	//INC1
    A_INC10 : BOOL ;	//INC10
    A_INC100 : BOOL ;	//INC100
    A_INC1000 : BOOL ;	//INC1000
    A_INC10000 : BOOL ;	//INC10000
    A_INCVar : BOOL ;	//INC variable
    f3 : BYTE ;
    E_MMC_AUTO : BOOL ;	//MMC Strobe AUTOMATIC mode
    E_MMC_MDA : BOOL ;	//MMC Strobe MDA mode
    E_MMC_JOG : BOOL ;	//MMC Strobe JOG mode
    f4_3 : BOOL ;
    f4_4 : BOOL ;
    f4_5 : BOOL ;
    f4_6 : BOOL ;
    f4_7 : BOOL ;
    E_MMC_TEACHIN : BOOL ;	//MMC Strobe machine function TEACH IN
    E_MMC_REPOS : BOOL ;	//MMC Strobe machine function REPOS
    E_MMC_REF : BOOL ;	//MMC Strobe Machine function REF
    f5_3 : BOOL ;
    f5_4 : BOOL ;
    f5_5 : BOOL ;
    f5_6 : BOOL ;
    f5_7 : BOOL ;
    E_AUTO : BOOL ;	//Active AUTOMATIC mode
    E_MDA : BOOL ;	//Active MDA mode
    E_JOG : BOOL ;	//Active JOG mode
    E_MGOK : BOOL ;	//Mode group ready
    E_MGreseted : BOOL ;	// Mode Group reseted
    E_NCKintJOG : BOOL ;	// NCK internal JOG active
    f6_6 : BOOL ;
    E_ChanReset : BOOL ;	//All channels in reset state
    E_TEACHIN : BOOL ;	//Active machine function TEACH IN
    E_REPOS : BOOL ;	//Active machine function REPOS
    E_REF : BOOL ;	//Active machine function REF
    f7_3 : BOOL ;
    f7_4 : BOOL ;
    f7_5 : BOOL ;
    f7_6 : BOOL ;
    f7_7 : BOOL ;
    E_INC1 : BOOL ;	//INC1
    E_INC10 : BOOL ;	//INC10
    E_INC100 : BOOL ;	//INC100
    E_INC1000 : BOOL ;	//INC1000
    E_INC10000 : BOOL ;	//INC10000
    E_INCVar : BOOL ;	//INC variable
    f8_6 : BOOL ;
    f8_7 : BOOL ;
    f9 : BYTE ;
    f10 : ARRAY  [10 .. 19 ] OF BYTE ;
   END_STRUCT ;
  END_STRUCT ;	
END_TYPE

